	calc8042: LREAL :=  10;
	calc8043: LREAL :=  10;
	calc8044: LREAL :=  10;
	calc8045: LREAL :=  10;
	calc8046: LREAL :=  10;
	calc8047: LREAL :=  10;
	calc8048: LREAL :=  10;
	calc8049: LREAL :=  10;
	calc8050: LREAL :=  10;
	calc8051: LREAL :=  10;
	calc8052: LREAL :=  10;
	calc8053: LREAL :=  10;
	calc8054: LREAL :=  10;
	calc8055: LREAL :=  10;
	calc8056: LREAL :=  10;
	calc8057: LREAL :=  10;
	calc8058: LREAL :=  10;
	calc8059: LREAL :=  10;
	calc8060: LREAL :=  10;
	calc8061: LREAL :=  10;
	calc8062: LREAL :=  10;
	calc8063: LREAL :=  10;
	calc8064: LREAL :=  10;
	calc8065: LREAL :=  10;
	calc8066: LREAL :=  10;
	calc8067: LREAL :=  10;
	calc8068: LREAL :=  10;
	calc8069: LREAL :=  10;
	calc8070: LREAL :=  10;
	calc8071: LREAL :=  10;
	calc8072: LREAL :=  10;
	calc8073: LREAL :=  10;
	calc8074: LREAL :=  10;
	calc8075: LREAL :=  10;
	calc8076: LREAL :=  10;
	calc8077: LREAL :=  10;
	calc8078: LREAL :=  10;
	calc8079: LREAL :=  10;
	calc8080: LREAL :=  10;
	calc8081: LREAL :=  10;
	calc8082: LREAL :=  10;
	calc8083: LREAL :=  10;
	calc8084: LREAL :=  10;
	calc8085: LREAL :=  10;
	calc8086: LREAL :=  10;
	calc8087: LREAL :=  10;
	calc8088: LREAL :=  10;
	calc8089: LREAL :=  10;
	calc8090: LREAL :=  10;
	calc8091: LREAL :=  10;
	calc8092: LREAL :=  10;
	calc8093: LREAL :=  10;
	calc8094: LREAL :=  10;
	calc8095: LREAL :=  10;
	calc8096: LREAL :=  10;
	calc8097: LREAL :=  10;
	calc8098: LREAL :=  10;
	calc8099: LREAL :=  10;
	calc8100: LREAL :=  10;
	calc8101: LREAL :=  10;
	calc8102: LREAL :=  10;
	calc8103: LREAL :=  10;
	calc8104: LREAL :=  10;
	calc8105: LREAL :=  10;
	calc8106: LREAL :=  10;
	calc8107: LREAL :=  10;
	calc8108: LREAL :=  10;
	calc8109: LREAL :=  10;
	calc8110: LREAL :=  10;
	calc8111: LREAL :=  10;
	calc8112: LREAL :=  10;
	calc8113: LREAL :=  10;
	calc8114: LREAL :=  10;
	calc8115: LREAL :=  10;
	calc8116: LREAL :=  10;
	calc8117: LREAL :=  10;
	calc8118: LREAL :=  10;
	calc8119: LREAL :=  10;
	calc8120: LREAL :=  10;
	calc8121: LREAL :=  10;
	calc8122: LREAL :=  10;
	calc8123: LREAL :=  10;
	calc8124: LREAL :=  10;
	calc8125: LREAL :=  10;
	calc8126: LREAL :=  10;
	calc8127: LREAL :=  10;
	calc8128: LREAL :=  10;
	calc8129: LREAL :=  10;
	calc8130: LREAL :=  10;
	calc8131: LREAL :=  10;
	calc8132: LREAL :=  10;
	calc8133: LREAL :=  10;
	calc8134: LREAL :=  10;
	calc8135: LREAL :=  10;
	calc8136: LREAL :=  10;
	calc8137: LREAL :=  10;
	calc8138: LREAL :=  10;
	calc8139: LREAL :=  10;
	calc8140: LREAL :=  10;
	calc8141: LREAL :=  10;
	calc8142: LREAL :=  10;
	calc8143: LREAL :=  10;
	calc8144: LREAL :=  10;
	calc8145: LREAL :=  10;
	calc8146: LREAL :=  10;
	calc8147: LREAL :=  10;
	calc8148: LREAL :=  10;
	calc8149: LREAL :=  10;
	calc8150: LREAL :=  10;
	calc8151: LREAL :=  10;
	calc8152: LREAL :=  10;
	calc8153: LREAL :=  10;
	calc8154: LREAL :=  10;
	calc8155: LREAL :=  10;
	calc8156: LREAL :=  10;
	calc8157: LREAL :=  10;
	calc8158: LREAL :=  10;
	calc8159: LREAL :=  10;
	calc8160: LREAL :=  10;
	calc8161: LREAL :=  10;
	calc8162: LREAL :=  10;
	calc8163: LREAL :=  10;
	calc8164: LREAL :=  10;
	calc8165: LREAL :=  10;
	calc8166: LREAL :=  10;
	calc8167: LREAL :=  10;
	calc8168: LREAL :=  10;
	calc8169: LREAL :=  10;
	calc8170: LREAL :=  10;
	calc8171: LREAL :=  10;
	calc8172: LREAL :=  10;
	calc8173: LREAL :=  10;
	calc8174: LREAL :=  10;
	calc8175: LREAL :=  10;
	calc8176: LREAL :=  10;
	calc8177: LREAL :=  10;
	calc8178: LREAL :=  10;
	calc8179: LREAL :=  10;
	calc8180: LREAL :=  10;
	calc8181: LREAL :=  10;
	calc8182: LREAL :=  10;
	calc8183: LREAL :=  10;
	calc8184: LREAL :=  10;
	calc8185: LREAL :=  10;
	calc8186: LREAL :=  10;
	calc8187: LREAL :=  10;
	calc8188: LREAL :=  10;
	calc8189: LREAL :=  10;
	calc8190: LREAL :=  10;
	calc8191: LREAL :=  10;
	calc8192: LREAL :=  10;
	calc8193: LREAL :=  10;
	calc8194: LREAL :=  10;
	calc8195: LREAL :=  10;
	calc8196: LREAL :=  10;
	calc8197: LREAL :=  10;
	calc8198: LREAL :=  10;
	calc8199: LREAL :=  10;
	calc8200: LREAL :=  10;
	calc8201: LREAL :=  10;
	calc8202: LREAL :=  10;
	calc8203: LREAL :=  10;
	calc8204: LREAL :=  10;
	calc8205: LREAL :=  10;
	calc8206: LREAL :=  10;
	calc8207: LREAL :=  10;
	calc8208: LREAL :=  10;
	calc8209: LREAL :=  10;
	calc8210: LREAL :=  10;
	calc8211: LREAL :=  10;
	calc8212: LREAL :=  10;
	calc8213: LREAL :=  10;
	calc8214: LREAL :=  10;
	calc8215: LREAL :=  10;
	calc8216: LREAL :=  10;
	calc8217: LREAL :=  10;
	calc8218: LREAL :=  10;
	calc8219: LREAL :=  10;
	calc8220: LREAL :=  10;
	calc8221: LREAL :=  10;
	calc8222: LREAL :=  10;
	calc8223: LREAL :=  10;
	calc8224: LREAL :=  10;
	calc8225: LREAL :=  10;
	calc8226: LREAL :=  10;
	calc8227: LREAL :=  10;
	calc8228: LREAL :=  10;
	calc8229: LREAL :=  10;
	calc8230: LREAL :=  10;
	calc8231: LREAL :=  10;
	calc8232: LREAL :=  10;
	calc8233: LREAL :=  10;
	calc8234: LREAL :=  10;
	calc8235: LREAL :=  10;
	calc8236: LREAL :=  10;
	calc8237: LREAL :=  10;
	calc8238: LREAL :=  10;
	calc8239: LREAL :=  10;
	calc8240: LREAL :=  10;
	calc8241: LREAL :=  10;
	calc8242: LREAL :=  10;
	calc8243: LREAL :=  10;
	calc8244: LREAL :=  10;
	calc8245: LREAL :=  10;
	calc8246: LREAL :=  10;
	calc8247: LREAL :=  10;
	calc8248: LREAL :=  10;
	calc8249: LREAL :=  10;
	calc8250: LREAL :=  10;
	calc8251: LREAL :=  10;
	calc8252: LREAL :=  10;
	calc8253: LREAL :=  10;
	calc8254: LREAL :=  10;
	calc8255: LREAL :=  10;
	calc8256: LREAL :=  10;
	calc8257: LREAL :=  10;
	calc8258: LREAL :=  10;
	calc8259: LREAL :=  10;
	calc8260: LREAL :=  10;
	calc8261: LREAL :=  10;
	calc8262: LREAL :=  10;
	calc8263: LREAL :=  10;
	calc8264: LREAL :=  10;
	calc8265: LREAL :=  10;
	calc8266: LREAL :=  10;
	calc8267: LREAL :=  10;
	calc8268: LREAL :=  10;
	calc8269: LREAL :=  10;
	calc8270: LREAL :=  10;
	calc8271: LREAL :=  10;
	calc8272: LREAL :=  10;
	calc8273: LREAL :=  10;
	calc8274: LREAL :=  10;
	calc8275: LREAL :=  10;
	calc8276: LREAL :=  10;
	calc8277: LREAL :=  10;
	calc8278: LREAL :=  10;
	calc8279: LREAL :=  10;
	calc8280: LREAL :=  10;
	calc8281: LREAL :=  10;
	calc8282: LREAL :=  10;
	calc8283: LREAL :=  10;
	calc8284: LREAL :=  10;
	calc8285: LREAL :=  10;
	calc8286: LREAL :=  10;
	calc8287: LREAL :=  10;
	calc8288: LREAL :=  10;
	calc8289: LREAL :=  10;
	calc8290: LREAL :=  10;
	calc8291: LREAL :=  10;
	calc8292: LREAL :=  10;
	calc8293: LREAL :=  10;
	calc8294: LREAL :=  10;
	calc8295: LREAL :=  10;
	calc8296: LREAL :=  10;
	calc8297: LREAL :=  10;
	calc8298: LREAL :=  10;
	calc8299: LREAL :=  10;
	calc8300: LREAL :=  10;
	calc8301: LREAL :=  10;
	calc8302: LREAL :=  10;
	calc8303: LREAL :=  10;
	calc8304: LREAL :=  10;
	calc8305: LREAL :=  10;
	calc8306: LREAL :=  10;
	calc8307: LREAL :=  10;
	calc8308: LREAL :=  10;
	calc8309: LREAL :=  10;
	calc8310: LREAL :=  10;
	calc8311: LREAL :=  10;
	calc8312: LREAL :=  10;
	calc8313: LREAL :=  10;
	calc8314: LREAL :=  10;
	calc8315: LREAL :=  10;
	calc8316: LREAL :=  10;
	calc8317: LREAL :=  10;
	calc8318: LREAL :=  10;
	calc8319: LREAL :=  10;
	calc8320: LREAL :=  10;
	calc8321: LREAL :=  10;
	calc8322: LREAL :=  10;
	calc8323: LREAL :=  10;
	calc8324: LREAL :=  10;
	calc8325: LREAL :=  10;
	calc8326: LREAL :=  10;
	calc8327: LREAL :=  10;
	calc8328: LREAL :=  10;
	calc8329: LREAL :=  10;
	calc8330: LREAL :=  10;
	calc8331: LREAL :=  10;
	calc8332: LREAL :=  10;
	calc8333: LREAL :=  10;
	calc8334: LREAL :=  10;
	calc8335: LREAL :=  10;
	calc8336: LREAL :=  10;
	calc8337: LREAL :=  10;
	calc8338: LREAL :=  10;
	calc8339: LREAL :=  10;
	calc8340: LREAL :=  10;
	calc8341: LREAL :=  10;
	calc8342: LREAL :=  10;
	calc8343: LREAL :=  10;
	calc8344: LREAL :=  10;
	calc8345: LREAL :=  10;
	calc8346: LREAL :=  10;
	calc8347: LREAL :=  10;
	calc8348: LREAL :=  10;
	calc8349: LREAL :=  10;
	calc8350: LREAL :=  10;
	calc8351: LREAL :=  10;
	calc8352: LREAL :=  10;
	calc8353: LREAL :=  10;
	calc8354: LREAL :=  10;
	calc8355: LREAL :=  10;
	calc8356: LREAL :=  10;
	calc8357: LREAL :=  10;
	calc8358: LREAL :=  10;
	calc8359: LREAL :=  10;
	calc8360: LREAL :=  10;
	calc8361: LREAL :=  10;
	calc8362: LREAL :=  10;
	calc8363: LREAL :=  10;
	calc8364: LREAL :=  10;
	calc8365: LREAL :=  10;
	calc8366: LREAL :=  10;
	calc8367: LREAL :=  10;
	calc8368: LREAL :=  10;
	calc8369: LREAL :=  10;
	calc8370: LREAL :=  10;
	calc8371: LREAL :=  10;
	calc8372: LREAL :=  10;
	calc8373: LREAL :=  10;
	calc8374: LREAL :=  10;
	calc8375: LREAL :=  10;
	calc8376: LREAL :=  10;
	calc8377: LREAL :=  10;
	calc8378: LREAL :=  10;
	calc8379: LREAL :=  10;
	calc8380: LREAL :=  10;
	calc8381: LREAL :=  10;
	calc8382: LREAL :=  10;
	calc8383: LREAL :=  10;
	calc8384: LREAL :=  10;
	calc8385: LREAL :=  10;
	calc8386: LREAL :=  10;
	calc8387: LREAL :=  10;
	calc8388: LREAL :=  10;
	calc8389: LREAL :=  10;
	calc8390: LREAL :=  10;
	calc8391: LREAL :=  10;
	calc8392: LREAL :=  10;
	calc8393: LREAL :=  10;
	calc8394: LREAL :=  10;
	calc8395: LREAL :=  10;
	calc8396: LREAL :=  10;
	calc8397: LREAL :=  10;
	calc8398: LREAL :=  10;
	calc8399: LREAL :=  10;
	calc8400: LREAL :=  10;
	calc8401: LREAL :=  10;
	calc8402: LREAL :=  10;
	calc8403: LREAL :=  10;
	calc8404: LREAL :=  10;
	calc8405: LREAL :=  10;
	calc8406: LREAL :=  10;
	calc8407: LREAL :=  10;
	calc8408: LREAL :=  10;
	calc8409: LREAL :=  10;
	calc8410: LREAL :=  10;
	calc8411: LREAL :=  10;
	calc8412: LREAL :=  10;
	calc8413: LREAL :=  10;
	calc8414: LREAL :=  10;
	calc8415: LREAL :=  10;
	calc8416: LREAL :=  10;
	calc8417: LREAL :=  10;
	calc8418: LREAL :=  10;
	calc8419: LREAL :=  10;
	calc8420: LREAL :=  10;
	calc8421: LREAL :=  10;
	calc8422: LREAL :=  10;
	calc8423: LREAL :=  10;
	calc8424: LREAL :=  10;
	calc8425: LREAL :=  10;
	calc8426: LREAL :=  10;
	calc8427: LREAL :=  10;
	calc8428: LREAL :=  10;
	calc8429: LREAL :=  10;
	calc8430: LREAL :=  10;
	calc8431: LREAL :=  10;
	calc8432: LREAL :=  10;
	calc8433: LREAL :=  10;
	calc8434: LREAL :=  10;
	calc8435: LREAL :=  10;
	calc8436: LREAL :=  10;
	calc8437: LREAL :=  10;
	calc8438: LREAL :=  10;
	calc8439: LREAL :=  10;
	calc8440: LREAL :=  10;
	calc8441: LREAL :=  10;
	calc8442: LREAL :=  10;
	calc8443: LREAL :=  10;
	calc8444: LREAL :=  10;
	calc8445: LREAL :=  10;
	calc8446: LREAL :=  10;
	calc8447: LREAL :=  10;
	calc8448: LREAL :=  10;
	calc8449: LREAL :=  10;
	calc8450: LREAL :=  10;
	calc8451: LREAL :=  10;
	calc8452: LREAL :=  10;
	calc8453: LREAL :=  10;
	calc8454: LREAL :=  10;
	calc8455: LREAL :=  10;
	calc8456: LREAL :=  10;
	calc8457: LREAL :=  10;
	calc8458: LREAL :=  10;
	calc8459: LREAL :=  10;
	calc8460: LREAL :=  10;
	calc8461: LREAL :=  10;
	calc8462: LREAL :=  10;
	calc8463: LREAL :=  10;
	calc8464: LREAL :=  10;
	calc8465: LREAL :=  10;
	calc8466: LREAL :=  10;
	calc8467: LREAL :=  10;
	calc8468: LREAL :=  10;
	calc8469: LREAL :=  10;
	calc8470: LREAL :=  10;
	calc8471: LREAL :=  10;
	calc8472: LREAL :=  10;
	calc8473: LREAL :=  10;
	calc8474: LREAL :=  10;
	calc8475: LREAL :=  10;
	calc8476: LREAL :=  10;
	calc8477: LREAL :=  10;
	calc8478: LREAL :=  10;
	calc8479: LREAL :=  10;
	calc8480: LREAL :=  10;
	calc8481: LREAL :=  10;
	calc8482: LREAL :=  10;
	calc8483: LREAL :=  10;
	calc8484: LREAL :=  10;
	calc8485: LREAL :=  10;
	calc8486: LREAL :=  10;
	calc8487: LREAL :=  10;
	calc8488: LREAL :=  10;
	calc8489: LREAL :=  10;
	calc8490: LREAL :=  10;
	calc8491: LREAL :=  10;
	calc8492: LREAL :=  10;
	calc8493: LREAL :=  10;
	calc8494: LREAL :=  10;
	calc8495: LREAL :=  10;
	calc8496: LREAL :=  10;
	calc8497: LREAL :=  10;
	calc8498: LREAL :=  10;
	calc8499: LREAL :=  10;
	calc8500: LREAL :=  10;
	calc8501: LREAL :=  10;
	calc8502: LREAL :=  10;
	calc8503: LREAL :=  10;
	calc8504: LREAL :=  10;
	calc8505: LREAL :=  10;
	calc8506: LREAL :=  10;
	calc8507: LREAL :=  10;
	calc8508: LREAL :=  10;
	calc8509: LREAL :=  10;
	calc8510: LREAL :=  10;
	calc8511: LREAL :=  10;
	calc8512: LREAL :=  10;
	calc8513: LREAL :=  10;
	calc8514: LREAL :=  10;
	calc8515: LREAL :=  10;
	calc8516: LREAL :=  10;
	calc8517: LREAL :=  10;
	calc8518: LREAL :=  10;
	calc8519: LREAL :=  10;
	calc8520: LREAL :=  10;
	calc8521: LREAL :=  10;
	calc8522: LREAL :=  10;
	calc8523: LREAL :=  10;
	calc8524: LREAL :=  10;
	calc8525: LREAL :=  10;
	calc8526: LREAL :=  10;
	calc8527: LREAL :=  10;
	calc8528: LREAL :=  10;
	calc8529: LREAL :=  10;
	calc8530: LREAL :=  10;
	calc8531: LREAL :=  10;
	calc8532: LREAL :=  10;
	calc8533: LREAL :=  10;
	calc8534: LREAL :=  10;
	calc8535: LREAL :=  10;
	calc8536: LREAL :=  10;
	calc8537: LREAL :=  10;
	calc8538: LREAL :=  10;
	calc8539: LREAL :=  10;
	calc8540: LREAL :=  10;
	calc8541: LREAL :=  10;
	calc8542: LREAL :=  10;
	calc8543: LREAL :=  10;
	calc8544: LREAL :=  10;
	calc8545: LREAL :=  10;
	calc8546: LREAL :=  10;
	calc8547: LREAL :=  10;
	calc8548: LREAL :=  10;
	calc8549: LREAL :=  10;
	calc8550: LREAL :=  10;
	calc8551: LREAL :=  10;
	calc8552: LREAL :=  10;
	calc8553: LREAL :=  10;
	calc8554: LREAL :=  10;
	calc8555: LREAL :=  10;
	calc8556: LREAL :=  10;
	calc8557: LREAL :=  10;
	calc8558: LREAL :=  10;
	calc8559: LREAL :=  10;
	calc8560: LREAL :=  10;
	calc8561: LREAL :=  10;
	calc8562: LREAL :=  10;
	calc8563: LREAL :=  10;
	calc8564: LREAL :=  10;
	calc8565: LREAL :=  10;
	calc8566: LREAL :=  10;
	calc8567: LREAL :=  10;
	calc8568: LREAL :=  10;
	calc8569: LREAL :=  10;
	calc8570: LREAL :=  10;
	calc8571: LREAL :=  10;
	calc8572: LREAL :=  10;
	calc8573: LREAL :=  10;
	calc8574: LREAL :=  10;
	calc8575: LREAL :=  10;
	calc8576: LREAL :=  10;
	calc8577: LREAL :=  10;
	calc8578: LREAL :=  10;
	calc8579: LREAL :=  10;
	calc8580: LREAL :=  10;
	calc8581: LREAL :=  10;
	calc8582: LREAL :=  10;
	calc8583: LREAL :=  10;
	calc8584: LREAL :=  10;
	calc8585: LREAL :=  10;
	calc8586: LREAL :=  10;
	calc8587: LREAL :=  10;
	calc8588: LREAL :=  10;
	calc8589: LREAL :=  10;
	calc8590: LREAL :=  10;
	calc8591: LREAL :=  10;
	calc8592: LREAL :=  10;
	calc8593: LREAL :=  10;
	calc8594: LREAL :=  10;
	calc8595: LREAL :=  10;
	calc8596: LREAL :=  10;
	calc8597: LREAL :=  10;
	calc8598: LREAL :=  10;
	calc8599: LREAL :=  10;
	calc8600: LREAL :=  10;
	calc8601: LREAL :=  10;
	calc8602: LREAL :=  10;
	calc8603: LREAL :=  10;
	calc8604: LREAL :=  10;
	calc8605: LREAL :=  10;
	calc8606: LREAL :=  10;
	calc8607: LREAL :=  10;
	calc8608: LREAL :=  10;
	calc8609: LREAL :=  10;
	calc8610: LREAL :=  10;
	calc8611: LREAL :=  10;
	calc8612: LREAL :=  10;
	calc8613: LREAL :=  10;
	calc8614: LREAL :=  10;
	calc8615: LREAL :=  10;
	calc8616: LREAL :=  10;
	calc8617: LREAL :=  10;
	calc8618: LREAL :=  10;
	calc8619: LREAL :=  10;
	calc8620: LREAL :=  10;
	calc8621: LREAL :=  10;
	calc8622: LREAL :=  10;
	calc8623: LREAL :=  10;
	calc8624: LREAL :=  10;
	calc8625: LREAL :=  10;
	calc8626: LREAL :=  10;
	calc8627: LREAL :=  10;
	calc8628: LREAL :=  10;
	calc8629: LREAL :=  10;
	calc8630: LREAL :=  10;
	calc8631: LREAL :=  10;
	calc8632: LREAL :=  10;
	calc8633: LREAL :=  10;
	calc8634: LREAL :=  10;
	calc8635: LREAL :=  10;
	calc8636: LREAL :=  10;
	calc8637: LREAL :=  10;
	calc8638: LREAL :=  10;
	calc8639: LREAL :=  10;
	calc8640: LREAL :=  10;
	calc8641: LREAL :=  10;
	calc8642: LREAL :=  10;
	calc8643: LREAL :=  10;
	calc8644: LREAL :=  10;
	calc8645: LREAL :=  10;
	calc8646: LREAL :=  10;
	calc8647: LREAL :=  10;
	calc8648: LREAL :=  10;
	calc8649: LREAL :=  10;
	calc8650: LREAL :=  10;
	calc8651: LREAL :=  10;
	calc8652: LREAL :=  10;
	calc8653: LREAL :=  10;
	calc8654: LREAL :=  10;
	calc8655: LREAL :=  10;
	calc8656: LREAL :=  10;
	calc8657: LREAL :=  10;
	calc8658: LREAL :=  10;
	calc8659: LREAL :=  10;
	calc8660: LREAL :=  10;
	calc8661: LREAL :=  10;
	calc8662: LREAL :=  10;
	calc8663: LREAL :=  10;
	calc8664: LREAL :=  10;
	calc8665: LREAL :=  10;
	calc8666: LREAL :=  10;
	calc8667: LREAL :=  10;
	calc8668: LREAL :=  10;
	calc8669: LREAL :=  10;
	calc8670: LREAL :=  10;
	calc8671: LREAL :=  10;
	calc8672: LREAL :=  10;
	calc8673: LREAL :=  10;
	calc8674: LREAL :=  10;
	calc8675: LREAL :=  10;
	calc8676: LREAL :=  10;
	calc8677: LREAL :=  10;
	calc8678: LREAL :=  10;
	calc8679: LREAL :=  10;
	calc8680: LREAL :=  10;
	calc8681: LREAL :=  10;
	calc8682: LREAL :=  10;
	calc8683: LREAL :=  10;
	calc8684: LREAL :=  10;
	calc8685: LREAL :=  10;
	calc8686: LREAL :=  10;
	calc8687: LREAL :=  10;
	calc8688: LREAL :=  10;
	calc8689: LREAL :=  10;
	calc8690: LREAL :=  10;
	calc8691: LREAL :=  10;
	calc8692: LREAL :=  10;
	calc8693: LREAL :=  10;
	calc8694: LREAL :=  10;
	calc8695: LREAL :=  10;
	calc8696: LREAL :=  10;
	calc8697: LREAL :=  10;
	calc8698: LREAL :=  10;
	calc8699: LREAL :=  10;
	calc8700: LREAL :=  10;
	calc8701: LREAL :=  10;
	calc8702: LREAL :=  10;
	calc8703: LREAL :=  10;
	calc8704: LREAL :=  10;
	calc8705: LREAL :=  10;
	calc8706: LREAL :=  10;
	calc8707: LREAL :=  10;
	calc8708: LREAL :=  10;
	calc8709: LREAL :=  10;
	calc8710: LREAL :=  10;
	calc8711: LREAL :=  10;
	calc8712: LREAL :=  10;
	calc8713: LREAL :=  10;
	calc8714: LREAL :=  10;
	calc8715: LREAL :=  10;
	calc8716: LREAL :=  10;
	calc8717: LREAL :=  10;
	calc8718: LREAL :=  10;
	calc8719: LREAL :=  10;
	calc8720: LREAL :=  10;
	calc8721: LREAL :=  10;
	calc8722: LREAL :=  10;
	calc8723: LREAL :=  10;
	calc8724: LREAL :=  10;
	calc8725: LREAL :=  10;
	calc8726: LREAL :=  10;
	calc8727: LREAL :=  10;
	calc8728: LREAL :=  10;
	calc8729: LREAL :=  10;
	calc8730: LREAL :=  10;
	calc8731: LREAL :=  10;
	calc8732: LREAL :=  10;
	calc8733: LREAL :=  10;
	calc8734: LREAL :=  10;
	calc8735: LREAL :=  10;
	calc8736: LREAL :=  10;
	calc8737: LREAL :=  10;
	calc8738: LREAL :=  10;
	calc8739: LREAL :=  10;
	calc8740: LREAL :=  10;
	calc8741: LREAL :=  10;
	calc8742: LREAL :=  10;
	calc8743: LREAL :=  10;
	calc8744: LREAL :=  10;
	calc8745: LREAL :=  10;
	calc8746: LREAL :=  10;
	calc8747: LREAL :=  10;
	calc8748: LREAL :=  10;
	calc8749: LREAL :=  10;
	calc8750: LREAL :=  10;
	calc8751: LREAL :=  10;
	calc8752: LREAL :=  10;
	calc8753: LREAL :=  10;
	calc8754: LREAL :=  10;
	calc8755: LREAL :=  10;
	calc8756: LREAL :=  10;
	calc8757: LREAL :=  10;
	calc8758: LREAL :=  10;
	calc8759: LREAL :=  10;
	calc8760: LREAL :=  10;
	calc8761: LREAL :=  10;
	calc8762: LREAL :=  10;
	calc8763: LREAL :=  10;
	calc8764: LREAL :=  10;
	calc8765: LREAL :=  10;
	calc8766: LREAL :=  10;
	calc8767: LREAL :=  10;
	calc8768: LREAL :=  10;
	calc8769: LREAL :=  10;
	calc8770: LREAL :=  10;
	calc8771: LREAL :=  10;
	calc8772: LREAL :=  10;
	calc8773: LREAL :=  10;
	calc8774: LREAL :=  10;
	calc8775: LREAL :=  10;
	calc8776: LREAL :=  10;
	calc8777: LREAL :=  10;
	calc8778: LREAL :=  10;
	calc8779: LREAL :=  10;
	calc8780: LREAL :=  10;
	calc8781: LREAL :=  10;
	calc8782: LREAL :=  10;
	calc8783: LREAL :=  10;
	calc8784: LREAL :=  10;
	calc8785: LREAL :=  10;
	calc8786: LREAL :=  10;
	calc8787: LREAL :=  10;
	calc8788: LREAL :=  10;
	calc8789: LREAL :=  10;
	calc8790: LREAL :=  10;
	calc8791: LREAL :=  10;
	calc8792: LREAL :=  10;
	calc8793: LREAL :=  10;
	calc8794: LREAL :=  10;
	calc8795: LREAL :=  10;
	calc8796: LREAL :=  10;
	calc8797: LREAL :=  10;
	calc8798: LREAL :=  10;
	calc8799: LREAL :=  10;
	calc8800: LREAL :=  10;
	calc8801: LREAL :=  10;
	calc8802: LREAL :=  10;
	calc8803: LREAL :=  10;
	calc8804: LREAL :=  10;
	calc8805: LREAL :=  10;
	calc8806: LREAL :=  10;
	calc8807: LREAL :=  10;
	calc8808: LREAL :=  10;
	calc8809: LREAL :=  10;
	calc8810: LREAL :=  10;
	calc8811: LREAL :=  10;
	calc8812: LREAL :=  10;
	calc8813: LREAL :=  10;
	calc8814: LREAL :=  10;
	calc8815: LREAL :=  10;
	calc8816: LREAL :=  10;
	calc8817: LREAL :=  10;
	calc8818: LREAL :=  10;
	calc8819: LREAL :=  10;
	calc8820: LREAL :=  10;
	calc8821: LREAL :=  10;
	calc8822: LREAL :=  10;
	calc8823: LREAL :=  10;
	calc8824: LREAL :=  10;
	calc8825: LREAL :=  10;
	calc8826: LREAL :=  10;
	calc8827: LREAL :=  10;
	calc8828: LREAL :=  10;
	calc8829: LREAL :=  10;
	calc8830: LREAL :=  10;
	calc8831: LREAL :=  10;
	calc8832: LREAL :=  10;
	calc8833: LREAL :=  10;
	calc8834: LREAL :=  10;
	calc8835: LREAL :=  10;
	calc8836: LREAL :=  10;
	calc8837: LREAL :=  10;
	calc8838: LREAL :=  10;
	calc8839: LREAL :=  10;
	calc8840: LREAL :=  10;
	calc8841: LREAL :=  10;
	calc8842: LREAL :=  10;
	calc8843: LREAL :=  10;
	calc8844: LREAL :=  10;
	calc8845: LREAL :=  10;
	calc8846: LREAL :=  10;
	calc8847: LREAL :=  10;
	calc8848: LREAL :=  10;
	calc8849: LREAL :=  10;
	calc8850: LREAL :=  10;
	calc8851: LREAL :=  10;
	calc8852: LREAL :=  10;
	calc8853: LREAL :=  10;
	calc8854: LREAL :=  10;
	calc8855: LREAL :=  10;
	calc8856: LREAL :=  10;
	calc8857: LREAL :=  10;
	calc8858: LREAL :=  10;
	calc8859: LREAL :=  10;
	calc8860: LREAL :=  10;
	calc8861: LREAL :=  10;
	calc8862: LREAL :=  10;
	calc8863: LREAL :=  10;
	calc8864: LREAL :=  10;
	calc8865: LREAL :=  10;
	calc8866: LREAL :=  10;
	calc8867: LREAL :=  10;
	calc8868: LREAL :=  10;
	calc8869: LREAL :=  10;
	calc8870: LREAL :=  10;
	calc8871: LREAL :=  10;
	calc8872: LREAL :=  10;
	calc8873: LREAL :=  10;
	calc8874: LREAL :=  10;
	calc8875: LREAL :=  10;
	calc8876: LREAL :=  10;
	calc8877: LREAL :=  10;
	calc8878: LREAL :=  10;
	calc8879: LREAL :=  10;
	calc8880: LREAL :=  10;
	calc8881: LREAL :=  10;
	calc8882: LREAL :=  10;
	calc8883: LREAL :=  10;
	calc8884: LREAL :=  10;
	calc8885: LREAL :=  10;
	calc8886: LREAL :=  10;
	calc8887: LREAL :=  10;
	calc8888: LREAL :=  10;
	calc8889: LREAL :=  10;
	calc8890: LREAL :=  10;
	calc8891: LREAL :=  10;
	calc8892: LREAL :=  10;
	calc8893: LREAL :=  10;
	calc8894: LREAL :=  10;
	calc8895: LREAL :=  10;
	calc8896: LREAL :=  10;
	calc8897: LREAL :=  10;
	calc8898: LREAL :=  10;
	calc8899: LREAL :=  10;
	calc8900: LREAL :=  10;
	calc8901: LREAL :=  10;
	calc8902: LREAL :=  10;
	calc8903: LREAL :=  10;
	calc8904: LREAL :=  10;
	calc8905: LREAL :=  10;
	calc8906: LREAL :=  10;
	calc8907: LREAL :=  10;
	calc8908: LREAL :=  10;
	calc8909: LREAL :=  10;
	calc8910: LREAL :=  10;
	calc8911: LREAL :=  10;
	calc8912: LREAL :=  10;
	calc8913: LREAL :=  10;
	calc8914: LREAL :=  10;
	calc8915: LREAL :=  10;
	calc8916: LREAL :=  10;
	calc8917: LREAL :=  10;
	calc8918: LREAL :=  10;
	calc8919: LREAL :=  10;
	calc8920: LREAL :=  10;
	calc8921: LREAL :=  10;
	calc8922: LREAL :=  10;
	calc8923: LREAL :=  10;
	calc8924: LREAL :=  10;
	calc8925: LREAL :=  10;
	calc8926: LREAL :=  10;
	calc8927: LREAL :=  10;
	calc8928: LREAL :=  10;
	calc8929: LREAL :=  10;
	calc8930: LREAL :=  10;
	calc8931: LREAL :=  10;
	calc8932: LREAL :=  10;
	calc8933: LREAL :=  10;
	calc8934: LREAL :=  10;
	calc8935: LREAL :=  10;
	calc8936: LREAL :=  10;
	calc8937: LREAL :=  10;
	calc8938: LREAL :=  10;
	calc8939: LREAL :=  10;
	calc8940: LREAL :=  10;
	calc8941: LREAL :=  10;
	calc8942: LREAL :=  10;
	calc8943: LREAL :=  10;
	calc8944: LREAL :=  10;
	calc8945: LREAL :=  10;
	calc8946: LREAL :=  10;
	calc8947: LREAL :=  10;
	calc8948: LREAL :=  10;
	calc8949: LREAL :=  10;
	calc8950: LREAL :=  10;
	calc8951: LREAL :=  10;
	calc8952: LREAL :=  10;
	calc8953: LREAL :=  10;
	calc8954: LREAL :=  10;
	calc8955: LREAL :=  10;
	calc8956: LREAL :=  10;
	calc8957: LREAL :=  10;
	calc8958: LREAL :=  10;
	calc8959: LREAL :=  10;
	calc8960: LREAL :=  10;
	calc8961: LREAL :=  10;
	calc8962: LREAL :=  10;
	calc8963: LREAL :=  10;
	calc8964: LREAL :=  10;
	calc8965: LREAL :=  10;
	calc8966: LREAL :=  10;
	calc8967: LREAL :=  10;
	calc8968: LREAL :=  10;
	calc8969: LREAL :=  10;
	calc8970: LREAL :=  10;
	calc8971: LREAL :=  10;
	calc8972: LREAL :=  10;
	calc8973: LREAL :=  10;
	calc8974: LREAL :=  10;
	calc8975: LREAL :=  10;
	calc8976: LREAL :=  10;
	calc8977: LREAL :=  10;
	calc8978: LREAL :=  10;
	calc8979: LREAL :=  10;
	calc8980: LREAL :=  10;
	calc8981: LREAL :=  10;
	calc8982: LREAL :=  10;
	calc8983: LREAL :=  10;
	calc8984: LREAL :=  10;
	calc8985: LREAL :=  10;
	calc8986: LREAL :=  10;
	calc8987: LREAL :=  10;
	calc8988: LREAL :=  10;
	calc8989: LREAL :=  10;
	calc8990: LREAL :=  10;
	calc8991: LREAL :=  10;
	calc8992: LREAL :=  10;
	calc8993: LREAL :=  10;
	calc8994: LREAL :=  10;
	calc8995: LREAL :=  10;
	calc8996: LREAL :=  10;
	calc8997: LREAL :=  10;
	calc8998: LREAL :=  10;
	calc8999: LREAL :=  10;
	calc9000: LREAL :=  10;
	calc9001: LREAL :=  10;
	calc9002: LREAL :=  10;
	calc9003: LREAL :=  10;
	calc9004: LREAL :=  10;
	calc9005: LREAL :=  10;
	calc9006: LREAL :=  10;
	calc9007: LREAL :=  10;
	calc9008: LREAL :=  10;
	calc9009: LREAL :=  10;
	calc9010: LREAL :=  10;
	calc9011: LREAL :=  10;
	calc9012: LREAL :=  10;
	calc9013: LREAL :=  10;
	calc9014: LREAL :=  10;
	calc9015: LREAL :=  10;
	calc9016: LREAL :=  10;
	calc9017: LREAL :=  10;
	calc9018: LREAL :=  10;
	calc9019: LREAL :=  10;
	calc9020: LREAL :=  10;
	calc9021: LREAL :=  10;
	calc9022: LREAL :=  10;
	calc9023: LREAL :=  10;
	calc9024: LREAL :=  10;
	calc9025: LREAL :=  10;
	calc9026: LREAL :=  10;
	calc9027: LREAL :=  10;
	calc9028: LREAL :=  10;
	calc9029: LREAL :=  10;
	calc9030: LREAL :=  10;
	calc9031: LREAL :=  10;
	calc9032: LREAL :=  10;
	calc9033: LREAL :=  10;
	calc9034: LREAL :=  10;
	calc9035: LREAL :=  10;
	calc9036: LREAL :=  10;
	calc9037: LREAL :=  10;
	calc9038: LREAL :=  10;
	calc9039: LREAL :=  10;
	calc9040: LREAL :=  10;
	calc9041: LREAL :=  10;
	calc9042: LREAL :=  10;
	calc9043: LREAL :=  10;
	calc9044: LREAL :=  10;
	calc9045: LREAL :=  10;
	calc9046: LREAL :=  10;
	calc9047: LREAL :=  10;
	calc9048: LREAL :=  10;
	calc9049: LREAL :=  10;
	calc9050: LREAL :=  10;
	calc9051: LREAL :=  10;
	calc9052: LREAL :=  10;
	calc9053: LREAL :=  10;
	calc9054: LREAL :=  10;
	calc9055: LREAL :=  10;
	calc9056: LREAL :=  10;
	calc9057: LREAL :=  10;
	calc9058: LREAL :=  10;
	calc9059: LREAL :=  10;
	calc9060: LREAL :=  10;
	calc9061: LREAL :=  10;
	calc9062: LREAL :=  10;
	calc9063: LREAL :=  10;
	calc9064: LREAL :=  10;
	calc9065: LREAL :=  10;
	calc9066: LREAL :=  10;
	calc9067: LREAL :=  10;
	calc9068: LREAL :=  10;
	calc9069: LREAL :=  10;
	calc9070: LREAL :=  10;
	calc9071: LREAL :=  10;
	calc9072: LREAL :=  10;
	calc9073: LREAL :=  10;
	calc9074: LREAL :=  10;
	calc9075: LREAL :=  10;
	calc9076: LREAL :=  10;
	calc9077: LREAL :=  10;
	calc9078: LREAL :=  10;
	calc9079: LREAL :=  10;
	calc9080: LREAL :=  10;
	calc9081: LREAL :=  10;
	calc9082: LREAL :=  10;
	calc9083: LREAL :=  10;
	calc9084: LREAL :=  10;
	calc9085: LREAL :=  10;
	calc9086: LREAL :=  10;
	calc9087: LREAL :=  10;
	calc9088: LREAL :=  10;
	calc9089: LREAL :=  10;
	calc9090: LREAL :=  10;
	calc9091: LREAL :=  10;
	calc9092: LREAL :=  10;
	calc9093: LREAL :=  10;
	calc9094: LREAL :=  10;
	calc9095: LREAL :=  10;
	calc9096: LREAL :=  10;
	calc9097: LREAL :=  10;
	calc9098: LREAL :=  10;
	calc9099: LREAL :=  10;
	calc9100: LREAL :=  10;
	calc9101: LREAL :=  10;
	calc9102: LREAL :=  10;
	calc9103: LREAL :=  10;
	calc9104: LREAL :=  10;
	calc9105: LREAL :=  10;
	calc9106: LREAL :=  10;
	calc9107: LREAL :=  10;
	calc9108: LREAL :=  10;
	calc9109: LREAL :=  10;
	calc9110: LREAL :=  10;
	calc9111: LREAL :=  10;
	calc9112: LREAL :=  10;
	calc9113: LREAL :=  10;
	calc9114: LREAL :=  10;
	calc9115: LREAL :=  10;
	calc9116: LREAL :=  10;
	calc9117: LREAL :=  10;
	calc9118: LREAL :=  10;
	calc9119: LREAL :=  10;
	calc9120: LREAL :=  10;
	calc9121: LREAL :=  10;
	calc9122: LREAL :=  10;
	calc9123: LREAL :=  10;
	calc9124: LREAL :=  10;
	calc9125: LREAL :=  10;
	calc9126: LREAL :=  10;
	calc9127: LREAL :=  10;
	calc9128: LREAL :=  10;
	calc9129: LREAL :=  10;
	calc9130: LREAL :=  10;
	calc9131: LREAL :=  10;
	calc9132: LREAL :=  10;
	calc9133: LREAL :=  10;
	calc9134: LREAL :=  10;
	calc9135: LREAL :=  10;
	calc9136: LREAL :=  10;
	calc9137: LREAL :=  10;
	calc9138: LREAL :=  10;
	calc9139: LREAL :=  10;
	calc9140: LREAL :=  10;
	calc9141: LREAL :=  10;
	calc9142: LREAL :=  10;
	calc9143: LREAL :=  10;
	calc9144: LREAL :=  10;
	calc9145: LREAL :=  10;
	calc9146: LREAL :=  10;
	calc9147: LREAL :=  10;
	calc9148: LREAL :=  10;
	calc9149: LREAL :=  10;
	calc9150: LREAL :=  10;
	calc9151: LREAL :=  10;
	calc9152: LREAL :=  10;
	calc9153: LREAL :=  10;
	calc9154: LREAL :=  10;
	calc9155: LREAL :=  10;
	calc9156: LREAL :=  10;
	calc9157: LREAL :=  10;
	calc9158: LREAL :=  10;
	calc9159: LREAL :=  10;
	calc9160: LREAL :=  10;
	calc9161: LREAL :=  10;
	calc9162: LREAL :=  10;
	calc9163: LREAL :=  10;
	calc9164: LREAL :=  10;
	calc9165: LREAL :=  10;
	calc9166: LREAL :=  10;
	calc9167: LREAL :=  10;
	calc9168: LREAL :=  10;
	calc9169: LREAL :=  10;
	calc9170: LREAL :=  10;
	calc9171: LREAL :=  10;
	calc9172: LREAL :=  10;
	calc9173: LREAL :=  10;
	calc9174: LREAL :=  10;
	calc9175: LREAL :=  10;
	calc9176: LREAL :=  10;
	calc9177: LREAL :=  10;
	calc9178: LREAL :=  10;
	calc9179: LREAL :=  10;
	calc9180: LREAL :=  10;
	calc9181: LREAL :=  10;
	calc9182: LREAL :=  10;
	calc9183: LREAL :=  10;
	calc9184: LREAL :=  10;
	calc9185: LREAL :=  10;
	calc9186: LREAL :=  10;
	calc9187: LREAL :=  10;
	calc9188: LREAL :=  10;
	calc9189: LREAL :=  10;
	calc9190: LREAL :=  10;
	calc9191: LREAL :=  10;
	calc9192: LREAL :=  10;
	calc9193: LREAL :=  10;
	calc9194: LREAL :=  10;
	calc9195: LREAL :=  10;
	calc9196: LREAL :=  10;
	calc9197: LREAL :=  10;
	calc9198: LREAL :=  10;
	calc9199: LREAL :=  10;
	calc9200: LREAL :=  10;
	calc9201: LREAL :=  10;
	calc9202: LREAL :=  10;
	calc9203: LREAL :=  10;
	calc9204: LREAL :=  10;
	calc9205: LREAL :=  10;
	calc9206: LREAL :=  10;
	calc9207: LREAL :=  10;
	calc9208: LREAL :=  10;
	calc9209: LREAL :=  10;
	calc9210: LREAL :=  10;
	calc9211: LREAL :=  10;
	calc9212: LREAL :=  10;
	calc9213: LREAL :=  10;
	calc9214: LREAL :=  10;
	calc9215: LREAL :=  10;
	calc9216: LREAL :=  10;
	calc9217: LREAL :=  10;
	calc9218: LREAL :=  10;
	calc9219: LREAL :=  10;
	calc9220: LREAL :=  10;
	calc9221: LREAL :=  10;
	calc9222: LREAL :=  10;
	calc9223: LREAL :=  10;
	calc9224: LREAL :=  10;
	calc9225: LREAL :=  10;
	calc9226: LREAL :=  10;
	calc9227: LREAL :=  10;
	calc9228: LREAL :=  10;
	calc9229: LREAL :=  10;
	calc9230: LREAL :=  10;
	calc9231: LREAL :=  10;
	calc9232: LREAL :=  10;
	calc9233: LREAL :=  10;
	calc9234: LREAL :=  10;
	calc9235: LREAL :=  10;
	calc9236: LREAL :=  10;
	calc9237: LREAL :=  10;
	calc9238: LREAL :=  10;
	calc9239: LREAL :=  10;
	calc9240: LREAL :=  10;
	calc9241: LREAL :=  10;
	calc9242: LREAL :=  10;
	calc9243: LREAL :=  10;
	calc9244: LREAL :=  10;
	calc9245: LREAL :=  10;
	calc9246: LREAL :=  10;
	calc9247: LREAL :=  10;
	calc9248: LREAL :=  10;
	calc9249: LREAL :=  10;
	calc9250: LREAL :=  10;
	calc9251: LREAL :=  10;
	calc9252: LREAL :=  10;
	calc9253: LREAL :=  10;
	calc9254: LREAL :=  10;
	calc9255: LREAL :=  10;
	calc9256: LREAL :=  10;
	calc9257: LREAL :=  10;
	calc9258: LREAL :=  10;
	calc9259: LREAL :=  10;
	calc9260: LREAL :=  10;
	calc9261: LREAL :=  10;
	calc9262: LREAL :=  10;
	calc9263: LREAL :=  10;
	calc9264: LREAL :=  10;
	calc9265: LREAL :=  10;
	calc9266: LREAL :=  10;
	calc9267: LREAL :=  10;
	calc9268: LREAL :=  10;
	calc9269: LREAL :=  10;
	calc9270: LREAL :=  10;
	calc9271: LREAL :=  10;
	calc9272: LREAL :=  10;
	calc9273: LREAL :=  10;
	calc9274: LREAL :=  10;
	calc9275: LREAL :=  10;
	calc9276: LREAL :=  10;
	calc9277: LREAL :=  10;
	calc9278: LREAL :=  10;
	calc9279: LREAL :=  10;
	calc9280: LREAL :=  10;
	calc9281: LREAL :=  10;
	calc9282: LREAL :=  10;
	calc9283: LREAL :=  10;
	calc9284: LREAL :=  10;
	calc9285: LREAL :=  10;
	calc9286: LREAL :=  10;
	calc9287: LREAL :=  10;
	calc9288: LREAL :=  10;
	calc9289: LREAL :=  10;
	calc9290: LREAL :=  10;
	calc9291: LREAL :=  10;
	calc9292: LREAL :=  10;
	calc9293: LREAL :=  10;
	calc9294: LREAL :=  10;
	calc9295: LREAL :=  10;
	calc9296: LREAL :=  10;
	calc9297: LREAL :=  10;
	calc9298: LREAL :=  10;
	calc9299: LREAL :=  10;
	calc9300: LREAL :=  10;
	calc9301: LREAL :=  10;
	calc9302: LREAL :=  10;
	calc9303: LREAL :=  10;
	calc9304: LREAL :=  10;
	calc9305: LREAL :=  10;
	calc9306: LREAL :=  10;
	calc9307: LREAL :=  10;
	calc9308: LREAL :=  10;
	calc9309: LREAL :=  10;
	calc9310: LREAL :=  10;
	calc9311: LREAL :=  10;
	calc9312: LREAL :=  10;
	calc9313: LREAL :=  10;
	calc9314: LREAL :=  10;
	calc9315: LREAL :=  10;
	calc9316: LREAL :=  10;
	calc9317: LREAL :=  10;
	calc9318: LREAL :=  10;
	calc9319: LREAL :=  10;
	calc9320: LREAL :=  10;
	calc9321: LREAL :=  10;
	calc9322: LREAL :=  10;
	calc9323: LREAL :=  10;
	calc9324: LREAL :=  10;
	calc9325: LREAL :=  10;
	calc9326: LREAL :=  10;
	calc9327: LREAL :=  10;
	calc9328: LREAL :=  10;
	calc9329: LREAL :=  10;
	calc9330: LREAL :=  10;
	calc9331: LREAL :=  10;
	calc9332: LREAL :=  10;
	calc9333: LREAL :=  10;
	calc9334: LREAL :=  10;
	calc9335: LREAL :=  10;
	calc9336: LREAL :=  10;
	calc9337: LREAL :=  10;
	calc9338: LREAL :=  10;
	calc9339: LREAL :=  10;
	calc9340: LREAL :=  10;
	calc9341: LREAL :=  10;
	calc9342: LREAL :=  10;
	calc9343: LREAL :=  10;
	calc9344: LREAL :=  10;
	calc9345: LREAL :=  10;
	calc9346: LREAL :=  10;
	calc9347: LREAL :=  10;
	calc9348: LREAL :=  10;
	calc9349: LREAL :=  10;
	calc9350: LREAL :=  10;
	calc9351: LREAL :=  10;
	calc9352: LREAL :=  10;
	calc9353: LREAL :=  10;
	calc9354: LREAL :=  10;
	calc9355: LREAL :=  10;
	calc9356: LREAL :=  10;
	calc9357: LREAL :=  10;
	calc9358: LREAL :=  10;
	calc9359: LREAL :=  10;
	calc9360: LREAL :=  10;
	calc9361: LREAL :=  10;
	calc9362: LREAL :=  10;
	calc9363: LREAL :=  10;
	calc9364: LREAL :=  10;
	calc9365: LREAL :=  10;
	calc9366: LREAL :=  10;
	calc9367: LREAL :=  10;
	calc9368: LREAL :=  10;
	calc9369: LREAL :=  10;
	calc9370: LREAL :=  10;
	calc9371: LREAL :=  10;
	calc9372: LREAL :=  10;
	calc9373: LREAL :=  10;
	calc9374: LREAL :=  10;
	calc9375: LREAL :=  10;
	calc9376: LREAL :=  10;
	calc9377: LREAL :=  10;
	calc9378: LREAL :=  10;
	calc9379: LREAL :=  10;
	calc9380: LREAL :=  10;
	calc9381: LREAL :=  10;
	calc9382: LREAL :=  10;
	calc9383: LREAL :=  10;
	calc9384: LREAL :=  10;
	calc9385: LREAL :=  10;
	calc9386: LREAL :=  10;
	calc9387: LREAL :=  10;
	calc9388: LREAL :=  10;
	calc9389: LREAL :=  10;
	calc9390: LREAL :=  10;
	calc9391: LREAL :=  10;
	calc9392: LREAL :=  10;
	calc9393: LREAL :=  10;
	calc9394: LREAL :=  10;
	calc9395: LREAL :=  10;
	calc9396: LREAL :=  10;
	calc9397: LREAL :=  10;
	calc9398: LREAL :=  10;
	calc9399: LREAL :=  10;
	calc9400: LREAL :=  10;
	calc9401: LREAL :=  10;
	calc9402: LREAL :=  10;
	calc9403: LREAL :=  10;
	calc9404: LREAL :=  10;
	calc9405: LREAL :=  10;
	calc9406: LREAL :=  10;
	calc9407: LREAL :=  10;
	calc9408: LREAL :=  10;
	calc9409: LREAL :=  10;
	calc9410: LREAL :=  10;
	calc9411: LREAL :=  10;
	calc9412: LREAL :=  10;
	calc9413: LREAL :=  10;
	calc9414: LREAL :=  10;
	calc9415: LREAL :=  10;
	calc9416: LREAL :=  10;
	calc9417: LREAL :=  10;
	calc9418: LREAL :=  10;
	calc9419: LREAL :=  10;
	calc9420: LREAL :=  10;
	calc9421: LREAL :=  10;
	calc9422: LREAL :=  10;
	calc9423: LREAL :=  10;
	calc9424: LREAL :=  10;
	calc9425: LREAL :=  10;
	calc9426: LREAL :=  10;
	calc9427: LREAL :=  10;
	calc9428: LREAL :=  10;
	calc9429: LREAL :=  10;
	calc9430: LREAL :=  10;
	calc9431: LREAL :=  10;
	calc9432: LREAL :=  10;
	calc9433: LREAL :=  10;
	calc9434: LREAL :=  10;
	calc9435: LREAL :=  10;
	calc9436: LREAL :=  10;
	calc9437: LREAL :=  10;
	calc9438: LREAL :=  10;
	calc9439: LREAL :=  10;
	calc9440: LREAL :=  10;
	calc9441: LREAL :=  10;
	calc9442: LREAL :=  10;
	calc9443: LREAL :=  10;
	calc9444: LREAL :=  10;
	calc9445: LREAL :=  10;
	calc9446: LREAL :=  10;
	calc9447: LREAL :=  10;
	calc9448: LREAL :=  10;
	calc9449: LREAL :=  10;
	calc9450: LREAL :=  10;
	calc9451: LREAL :=  10;
	calc9452: LREAL :=  10;
	calc9453: LREAL :=  10;
	calc9454: LREAL :=  10;
	calc9455: LREAL :=  10;
	calc9456: LREAL :=  10;
	calc9457: LREAL :=  10;
	calc9458: LREAL :=  10;
	calc9459: LREAL :=  10;
	calc9460: LREAL :=  10;
	calc9461: LREAL :=  10;
	calc9462: LREAL :=  10;
	calc9463: LREAL :=  10;
	calc9464: LREAL :=  10;
	calc9465: LREAL :=  10;
	calc9466: LREAL :=  10;
	calc9467: LREAL :=  10;
	calc9468: LREAL :=  10;
	calc9469: LREAL :=  10;
	calc9470: LREAL :=  10;
	calc9471: LREAL :=  10;
	calc9472: LREAL :=  10;
	calc9473: LREAL :=  10;
	calc9474: LREAL :=  10;
	calc9475: LREAL :=  10;
	calc9476: LREAL :=  10;
	calc9477: LREAL :=  10;
	calc9478: LREAL :=  10;
	calc9479: LREAL :=  10;
	calc9480: LREAL :=  10;
	calc9481: LREAL :=  10;
	calc9482: LREAL :=  10;
	calc9483: LREAL :=  10;
	calc9484: LREAL :=  10;
	calc9485: LREAL :=  10;
	calc9486: LREAL :=  10;
	calc9487: LREAL :=  10;
	calc9488: LREAL :=  10;
	calc9489: LREAL :=  10;
	calc9490: LREAL :=  10;
	calc9491: LREAL :=  10;
	calc9492: LREAL :=  10;
	calc9493: LREAL :=  10;
	calc9494: LREAL :=  10;
	calc9495: LREAL :=  10;
	calc9496: LREAL :=  10;
	calc9497: LREAL :=  10;
	calc9498: LREAL :=  10;
	calc9499: LREAL :=  10;
	calc9500: LREAL :=  10;
	calc9501: LREAL :=  10;
	calc9502: LREAL :=  10;
	calc9503: LREAL :=  10;
	calc9504: LREAL :=  10;
	calc9505: LREAL :=  10;
	calc9506: LREAL :=  10;
	calc9507: LREAL :=  10;
	calc9508: LREAL :=  10;
	calc9509: LREAL :=  10;
	calc9510: LREAL :=  10;
	calc9511: LREAL :=  10;
	calc9512: LREAL :=  10;
	calc9513: LREAL :=  10;
	calc9514: LREAL :=  10;
	calc9515: LREAL :=  10;
	calc9516: LREAL :=  10;
	calc9517: LREAL :=  10;
	calc9518: LREAL :=  10;
	calc9519: LREAL :=  10;
	calc9520: LREAL :=  10;
	calc9521: LREAL :=  10;
	calc9522: LREAL :=  10;
	calc9523: LREAL :=  10;
	calc9524: LREAL :=  10;
	calc9525: LREAL :=  10;
	calc9526: LREAL :=  10;
	calc9527: LREAL :=  10;
	calc9528: LREAL :=  10;
	calc9529: LREAL :=  10;
	calc9530: LREAL :=  10;
	calc9531: LREAL :=  10;
	calc9532: LREAL :=  10;
	calc9533: LREAL :=  10;
	calc9534: LREAL :=  10;
	calc9535: LREAL :=  10;
	calc9536: LREAL :=  10;
	calc9537: LREAL :=  10;
	calc9538: LREAL :=  10;
	calc9539: LREAL :=  10;
	calc9540: LREAL :=  10;
	calc9541: LREAL :=  10;
	calc9542: LREAL :=  10;
	calc9543: LREAL :=  10;
	calc9544: LREAL :=  10;
	calc9545: LREAL :=  10;
	calc9546: LREAL :=  10;
	calc9547: LREAL :=  10;
	calc9548: LREAL :=  10;
	calc9549: LREAL :=  10;
	calc9550: LREAL :=  10;
	calc9551: LREAL :=  10;
	calc9552: LREAL :=  10;
	calc9553: LREAL :=  10;
	calc9554: LREAL :=  10;
	calc9555: LREAL :=  10;
	calc9556: LREAL :=  10;
	calc9557: LREAL :=  10;
	calc9558: LREAL :=  10;
	calc9559: LREAL :=  10;
	calc9560: LREAL :=  10;
	calc9561: LREAL :=  10;
	calc9562: LREAL :=  10;
	calc9563: LREAL :=  10;
	calc9564: LREAL :=  10;
	calc9565: LREAL :=  10;
	calc9566: LREAL :=  10;
	calc9567: LREAL :=  10;
	calc9568: LREAL :=  10;
	calc9569: LREAL :=  10;
	calc9570: LREAL :=  10;
	calc9571: LREAL :=  10;
	calc9572: LREAL :=  10;
	calc9573: LREAL :=  10;
	calc9574: LREAL :=  10;
	calc9575: LREAL :=  10;
	calc9576: LREAL :=  10;
	calc9577: LREAL :=  10;
	calc9578: LREAL :=  10;
	calc9579: LREAL :=  10;
	calc9580: LREAL :=  10;
	calc9581: LREAL :=  10;
	calc9582: LREAL :=  10;
	calc9583: LREAL :=  10;
	calc9584: LREAL :=  10;
	calc9585: LREAL :=  10;
	calc9586: LREAL :=  10;
	calc9587: LREAL :=  10;
	calc9588: LREAL :=  10;
	calc9589: LREAL :=  10;
	calc9590: LREAL :=  10;
	calc9591: LREAL :=  10;
	calc9592: LREAL :=  10;
	calc9593: LREAL :=  10;
	calc9594: LREAL :=  10;
	calc9595: LREAL :=  10;
	calc9596: LREAL :=  10;
	calc9597: LREAL :=  10;
	calc9598: LREAL :=  10;
	calc9599: LREAL :=  10;
	calc9600: LREAL :=  10;
	calc9601: LREAL :=  10;
	calc9602: LREAL :=  10;
	calc9603: LREAL :=  10;
	calc9604: LREAL :=  10;
	calc9605: LREAL :=  10;
	calc9606: LREAL :=  10;
	calc9607: LREAL :=  10;
	calc9608: LREAL :=  10;
	calc9609: LREAL :=  10;
	calc9610: LREAL :=  10;
	calc9611: LREAL :=  10;
	calc9612: LREAL :=  10;
	calc9613: LREAL :=  10;
	calc9614: LREAL :=  10;
	calc9615: LREAL :=  10;
	calc9616: LREAL :=  10;
	calc9617: LREAL :=  10;
	calc9618: LREAL :=  10;
	calc9619: LREAL :=  10;
	calc9620: LREAL :=  10;
	calc9621: LREAL :=  10;
	calc9622: LREAL :=  10;
	calc9623: LREAL :=  10;
	calc9624: LREAL :=  10;
	calc9625: LREAL :=  10;
	calc9626: LREAL :=  10;
	calc9627: LREAL :=  10;
	calc9628: LREAL :=  10;
	calc9629: LREAL :=  10;
	calc9630: LREAL :=  10;
	calc9631: LREAL :=  10;
	calc9632: LREAL :=  10;
	calc9633: LREAL :=  10;
	calc9634: LREAL :=  10;
	calc9635: LREAL :=  10;
	calc9636: LREAL :=  10;
	calc9637: LREAL :=  10;
	calc9638: LREAL :=  10;
	calc9639: LREAL :=  10;
	calc9640: LREAL :=  10;
	calc9641: LREAL :=  10;
	calc9642: LREAL :=  10;
	calc9643: LREAL :=  10;
	calc9644: LREAL :=  10;
	calc9645: LREAL :=  10;
	calc9646: LREAL :=  10;
	calc9647: LREAL :=  10;
	calc9648: LREAL :=  10;
	calc9649: LREAL :=  10;
	calc9650: LREAL :=  10;
	calc9651: LREAL :=  10;
	calc9652: LREAL :=  10;
	calc9653: LREAL :=  10;
	calc9654: LREAL :=  10;
	calc9655: LREAL :=  10;
	calc9656: LREAL :=  10;
	calc9657: LREAL :=  10;
	calc9658: LREAL :=  10;
	calc9659: LREAL :=  10;
	calc9660: LREAL :=  10;
	calc9661: LREAL :=  10;
	calc9662: LREAL :=  10;
	calc9663: LREAL :=  10;
	calc9664: LREAL :=  10;
	calc9665: LREAL :=  10;
	calc9666: LREAL :=  10;
	calc9667: LREAL :=  10;
	calc9668: LREAL :=  10;
	calc9669: LREAL :=  10;
	calc9670: LREAL :=  10;
	calc9671: LREAL :=  10;
	calc9672: LREAL :=  10;
	calc9673: LREAL :=  10;
	calc9674: LREAL :=  10;
	calc9675: LREAL :=  10;
	calc9676: LREAL :=  10;
	calc9677: LREAL :=  10;
	calc9678: LREAL :=  10;
	calc9679: LREAL :=  10;
	calc9680: LREAL :=  10;
	calc9681: LREAL :=  10;
	calc9682: LREAL :=  10;
	calc9683: LREAL :=  10;
	calc9684: LREAL :=  10;
	calc9685: LREAL :=  10;
	calc9686: LREAL :=  10;
	calc9687: LREAL :=  10;
	calc9688: LREAL :=  10;
	calc9689: LREAL :=  10;
	calc9690: LREAL :=  10;
	calc9691: LREAL :=  10;
	calc9692: LREAL :=  10;
	calc9693: LREAL :=  10;
	calc9694: LREAL :=  10;
	calc9695: LREAL :=  10;
	calc9696: LREAL :=  10;
	calc9697: LREAL :=  10;
	calc9698: LREAL :=  10;
	calc9699: LREAL :=  10;
	calc9700: LREAL :=  10;
	calc9701: LREAL :=  10;
	calc9702: LREAL :=  10;
	calc9703: LREAL :=  10;
	calc9704: LREAL :=  10;
	calc9705: LREAL :=  10;
	calc9706: LREAL :=  10;
	calc9707: LREAL :=  10;
	calc9708: LREAL :=  10;
	calc9709: LREAL :=  10;
	calc9710: LREAL :=  10;
	calc9711: LREAL :=  10;
	calc9712: LREAL :=  10;
	calc9713: LREAL :=  10;
	calc9714: LREAL :=  10;
	calc9715: LREAL :=  10;
	calc9716: LREAL :=  10;
	calc9717: LREAL :=  10;
	calc9718: LREAL :=  10;
	calc9719: LREAL :=  10;
	calc9720: LREAL :=  10;
	calc9721: LREAL :=  10;
	calc9722: LREAL :=  10;
	calc9723: LREAL :=  10;
	calc9724: LREAL :=  10;
	calc9725: LREAL :=  10;
	calc9726: LREAL :=  10;
	calc9727: LREAL :=  10;
	calc9728: LREAL :=  10;
	calc9729: LREAL :=  10;
	calc9730: LREAL :=  10;
	calc9731: LREAL :=  10;
	calc9732: LREAL :=  10;
	calc9733: LREAL :=  10;
	calc9734: LREAL :=  10;
	calc9735: LREAL :=  10;
	calc9736: LREAL :=  10;
	calc9737: LREAL :=  10;
	calc9738: LREAL :=  10;
	calc9739: LREAL :=  10;
	calc9740: LREAL :=  10;
	calc9741: LREAL :=  10;
	calc9742: LREAL :=  10;
	calc9743: LREAL :=  10;
	calc9744: LREAL :=  10;
	calc9745: LREAL :=  10;
	calc9746: LREAL :=  10;
	calc9747: LREAL :=  10;
	calc9748: LREAL :=  10;
	calc9749: LREAL :=  10;
	calc9750: LREAL :=  10;
	calc9751: LREAL :=  10;
	calc9752: LREAL :=  10;
	calc9753: LREAL :=  10;
	calc9754: LREAL :=  10;
	calc9755: LREAL :=  10;
	calc9756: LREAL :=  10;
	calc9757: LREAL :=  10;
	calc9758: LREAL :=  10;
	calc9759: LREAL :=  10;
	calc9760: LREAL :=  10;
	calc9761: LREAL :=  10;
	calc9762: LREAL :=  10;
	calc9763: LREAL :=  10;
	calc9764: LREAL :=  10;
	calc9765: LREAL :=  10;
	calc9766: LREAL :=  10;
	calc9767: LREAL :=  10;
	calc9768: LREAL :=  10;
	calc9769: LREAL :=  10;
	calc9770: LREAL :=  10;
	calc9771: LREAL :=  10;
	calc9772: LREAL :=  10;
	calc9773: LREAL :=  10;
	calc9774: LREAL :=  10;
	calc9775: LREAL :=  10;
	calc9776: LREAL :=  10;
	calc9777: LREAL :=  10;
	calc9778: LREAL :=  10;
	calc9779: LREAL :=  10;
	calc9780: LREAL :=  10;
	calc9781: LREAL :=  10;
	calc9782: LREAL :=  10;
	calc9783: LREAL :=  10;
	calc9784: LREAL :=  10;
	calc9785: LREAL :=  10;
	calc9786: LREAL :=  10;
	calc9787: LREAL :=  10;
	calc9788: LREAL :=  10;
	calc9789: LREAL :=  10;
	calc9790: LREAL :=  10;
	calc9791: LREAL :=  10;
	calc9792: LREAL :=  10;
	calc9793: LREAL :=  10;
	calc9794: LREAL :=  10;
	calc9795: LREAL :=  10;
	calc9796: LREAL :=  10;
	calc9797: LREAL :=  10;
	calc9798: LREAL :=  10;
	calc9799: LREAL :=  10;
	calc9800: LREAL :=  10;
	calc9801: LREAL :=  10;
	calc9802: LREAL :=  10;
	calc9803: LREAL :=  10;
	calc9804: LREAL :=  10;
	calc9805: LREAL :=  10;
	calc9806: LREAL :=  10;
	calc9807: LREAL :=  10;
	calc9808: LREAL :=  10;
	calc9809: LREAL :=  10;
	calc9810: LREAL :=  10;
	calc9811: LREAL :=  10;
	calc9812: LREAL :=  10;
	calc9813: LREAL :=  10;
	calc9814: LREAL :=  10;
	calc9815: LREAL :=  10;
	calc9816: LREAL :=  10;
	calc9817: LREAL :=  10;
	calc9818: LREAL :=  10;
	calc9819: LREAL :=  10;
	calc9820: LREAL :=  10;
	calc9821: LREAL :=  10;
	calc9822: LREAL :=  10;
	calc9823: LREAL :=  10;
	calc9824: LREAL :=  10;
	calc9825: LREAL :=  10;
	calc9826: LREAL :=  10;
	calc9827: LREAL :=  10;
	calc9828: LREAL :=  10;
	calc9829: LREAL :=  10;
	calc9830: LREAL :=  10;
	calc9831: LREAL :=  10;
	calc9832: LREAL :=  10;
	calc9833: LREAL :=  10;
	calc9834: LREAL :=  10;
	calc9835: LREAL :=  10;
	calc9836: LREAL :=  10;
	calc9837: LREAL :=  10;
	calc9838: LREAL :=  10;
	calc9839: LREAL :=  10;
	calc9840: LREAL :=  10;
	calc9841: LREAL :=  10;
	calc9842: LREAL :=  10;
	calc9843: LREAL :=  10;
	calc9844: LREAL :=  10;
	calc9845: LREAL :=  10;
	calc9846: LREAL :=  10;
	calc9847: LREAL :=  10;
	calc9848: LREAL :=  10;
	calc9849: LREAL :=  10;
	calc9850: LREAL :=  10;
	calc9851: LREAL :=  10;
	calc9852: LREAL :=  10;
	calc9853: LREAL :=  10;
	calc9854: LREAL :=  10;
	calc9855: LREAL :=  10;
	calc9856: LREAL :=  10;
	calc9857: LREAL :=  10;
	calc9858: LREAL :=  10;
	calc9859: LREAL :=  10;
	calc9860: LREAL :=  10;
	calc9861: LREAL :=  10;
	calc9862: LREAL :=  10;
	calc9863: LREAL :=  10;
	calc9864: LREAL :=  10;
	calc9865: LREAL :=  10;
	calc9866: LREAL :=  10;
	calc9867: LREAL :=  10;
	calc9868: LREAL :=  10;
	calc9869: LREAL :=  10;
	calc9870: LREAL :=  10;
	calc9871: LREAL :=  10;
	calc9872: LREAL :=  10;
	calc9873: LREAL :=  10;
	calc9874: LREAL :=  10;
	calc9875: LREAL :=  10;
	calc9876: LREAL :=  10;
	calc9877: LREAL :=  10;
	calc9878: LREAL :=  10;
	calc9879: LREAL :=  10;
	calc9880: LREAL :=  10;
	calc9881: LREAL :=  10;
	calc9882: LREAL :=  10;
	calc9883: LREAL :=  10;
	calc9884: LREAL :=  10;
	calc9885: LREAL :=  10;
	calc9886: LREAL :=  10;
	calc9887: LREAL :=  10;
	calc9888: LREAL :=  10;
	calc9889: LREAL :=  10;
	calc9890: LREAL :=  10;
	calc9891: LREAL :=  10;
	calc9892: LREAL :=  10;
	calc9893: LREAL :=  10;
	calc9894: LREAL :=  10;
	calc9895: LREAL :=  10;
	calc9896: LREAL :=  10;
	calc9897: LREAL :=  10;
	calc9898: LREAL :=  10;
	calc9899: LREAL :=  10;
	calc9900: LREAL :=  10;
	calc9901: LREAL :=  10;
	calc9902: LREAL :=  10;
	calc9903: LREAL :=  10;
	calc9904: LREAL :=  10;
	calc9905: LREAL :=  10;
	calc9906: LREAL :=  10;
	calc9907: LREAL :=  10;
	calc9908: LREAL :=  10;
	calc9909: LREAL :=  10;
	calc9910: LREAL :=  10;
	calc9911: LREAL :=  10;
	calc9912: LREAL :=  10;
	calc9913: LREAL :=  10;
	calc9914: LREAL :=  10;
	calc9915: LREAL :=  10;
	calc9916: LREAL :=  10;
	calc9917: LREAL :=  10;
	calc9918: LREAL :=  10;
	calc9919: LREAL :=  10;
	calc9920: LREAL :=  10;
	calc9921: LREAL :=  10;
	calc9922: LREAL :=  10;
	calc9923: LREAL :=  10;
	calc9924: LREAL :=  10;
	calc9925: LREAL :=  10;
	calc9926: LREAL :=  10;
	calc9927: LREAL :=  10;
	calc9928: LREAL :=  10;
	calc9929: LREAL :=  10;
	calc9930: LREAL :=  10;
	calc9931: LREAL :=  10;
	calc9932: LREAL :=  10;
	calc9933: LREAL :=  10;
	calc9934: LREAL :=  10;
	calc9935: LREAL :=  10;
	calc9936: LREAL :=  10;
	calc9937: LREAL :=  10;
	calc9938: LREAL :=  10;
	calc9939: LREAL :=  10;
	calc9940: LREAL :=  10;
	calc9941: LREAL :=  10;
	calc9942: LREAL :=  10;
	calc9943: LREAL :=  10;
	calc9944: LREAL :=  10;
	calc9945: LREAL :=  10;
	calc9946: LREAL :=  10;
	calc9947: LREAL :=  10;
	calc9948: LREAL :=  10;
	calc9949: LREAL :=  10;
	calc9950: LREAL :=  10;
	calc9951: LREAL :=  10;
	calc9952: LREAL :=  10;
	calc9953: LREAL :=  10;
	calc9954: LREAL :=  10;
	calc9955: LREAL :=  10;
	calc9956: LREAL :=  10;
	calc9957: LREAL :=  10;
	calc9958: LREAL :=  10;
	calc9959: LREAL :=  10;
	calc9960: LREAL :=  10;
	calc9961: LREAL :=  10;
	calc9962: LREAL :=  10;
	calc9963: LREAL :=  10;
	calc9964: LREAL :=  10;
	calc9965: LREAL :=  10;
	calc9966: LREAL :=  10;
	calc9967: LREAL :=  10;
	calc9968: LREAL :=  10;
	calc9969: LREAL :=  10;
	calc9970: LREAL :=  10;
	calc9971: LREAL :=  10;
	calc9972: LREAL :=  10;
	calc9973: LREAL :=  10;
	calc9974: LREAL :=  10;
	calc9975: LREAL :=  10;
	calc9976: LREAL :=  10;
	calc9977: LREAL :=  10;
	calc9978: LREAL :=  10;
	calc9979: LREAL :=  10;
	calc9980: LREAL :=  10;
	calc9981: LREAL :=  10;
	calc9982: LREAL :=  10;
	calc9983: LREAL :=  10;
	calc9984: LREAL :=  10;
	calc9985: LREAL :=  10;
	calc9986: LREAL :=  10;
	calc9987: LREAL :=  10;
	calc9988: LREAL :=  10;
	calc9989: LREAL :=  10;
	calc9990: LREAL :=  10;
	calc9991: LREAL :=  10;
	calc9992: LREAL :=  10;
	calc9993: LREAL :=  10;
	calc9994: LREAL :=  10;
	calc9995: LREAL :=  10;
	calc9996: LREAL :=  10;
	calc9997: LREAL :=  10;
	calc9998: LREAL :=  10;
	calc9999: LREAL :=  10;
	
		counter0: LREAL :=  0;
	counter1: LREAL :=  0;
	counter2: LREAL :=  0;
	counter3: LREAL :=  0;
	counter4: LREAL :=  0;
	counter5: LREAL :=  0;
	counter6: LREAL :=  0;
	counter7: LREAL :=  0;
	counter8: LREAL :=  0;
	counter9: LREAL :=  0;
	counter10: LREAL :=  0;
	counter11: LREAL :=  0;
	counter12: LREAL :=  0;
	counter13: LREAL :=  0;
	counter14: LREAL :=  0;
	counter15: LREAL :=  0;
	counter16: LREAL :=  0;
	counter17: LREAL :=  0;
	counter18: LREAL :=  0;
	counter19: LREAL :=  0;
	counter20: LREAL :=  0;
	counter21: LREAL :=  0;
	counter22: LREAL :=  0;
	counter23: LREAL :=  0;
	counter24: LREAL :=  0;
	counter25: LREAL :=  0;
	counter26: LREAL :=  0;
	counter27: LREAL :=  0;
	counter28: LREAL :=  0;
	counter29: LREAL :=  0;
	counter30: LREAL :=  0;
	counter31: LREAL :=  0;
	counter32: LREAL :=  0;
	counter33: LREAL :=  0;
	counter34: LREAL :=  0;
	counter35: LREAL :=  0;
	counter36: LREAL :=  0;
	counter37: LREAL :=  0;
	counter38: LREAL :=  0;
	counter39: LREAL :=  0;
	counter40: LREAL :=  0;
	counter41: LREAL :=  0;
	counter42: LREAL :=  0;
	counter43: LREAL :=  0;
	counter44: LREAL :=  0;
	counter45: LREAL :=  0;
	counter46: LREAL :=  0;
	counter47: LREAL :=  0;
	counter48: LREAL :=  0;
	counter49: LREAL :=  0;
	counter50: LREAL :=  0;
	counter51: LREAL :=  0;
	counter52: LREAL :=  0;
	counter53: LREAL :=  0;
	counter54: LREAL :=  0;
	counter55: LREAL :=  0;
	counter56: LREAL :=  0;
	counter57: LREAL :=  0;
	counter58: LREAL :=  0;
	counter59: LREAL :=  0;
	counter60: LREAL :=  0;
	counter61: LREAL :=  0;
	counter62: LREAL :=  0;
	counter63: LREAL :=  0;
	counter64: LREAL :=  0;
	counter65: LREAL :=  0;
	counter66: LREAL :=  0;
	counter67: LREAL :=  0;
	counter68: LREAL :=  0;
	counter69: LREAL :=  0;
	counter70: LREAL :=  0;
	counter71: LREAL :=  0;
	counter72: LREAL :=  0;
	counter73: LREAL :=  0;
	counter74: LREAL :=  0;
	counter75: LREAL :=  0;
	counter76: LREAL :=  0;
	counter77: LREAL :=  0;
	counter78: LREAL :=  0;
	counter79: LREAL :=  0;
	counter80: LREAL :=  0;
	counter81: LREAL :=  0;
	counter82: LREAL :=  0;
	counter83: LREAL :=  0;
	counter84: LREAL :=  0;
	counter85: LREAL :=  0;
	counter86: LREAL :=  0;
	counter87: LREAL :=  0;
	counter88: LREAL :=  0;
	counter89: LREAL :=  0;
	counter90: LREAL :=  0;
	counter91: LREAL :=  0;
	counter92: LREAL :=  0;
	counter93: LREAL :=  0;
	counter94: LREAL :=  0;
	counter95: LREAL :=  0;
	counter96: LREAL :=  0;
	counter97: LREAL :=  0;
	counter98: LREAL :=  0;
	counter99: LREAL :=  0;
	counter100: LREAL :=  0;
	counter101: LREAL :=  0;
	counter102: LREAL :=  0;
	counter103: LREAL :=  0;
	counter104: LREAL :=  0;
	counter105: LREAL :=  0;
	counter106: LREAL :=  0;
	counter107: LREAL :=  0;
	counter108: LREAL :=  0;
	counter109: LREAL :=  0;
	counter110: LREAL :=  0;
	counter111: LREAL :=  0;
	counter112: LREAL :=  0;
	counter113: LREAL :=  0;
	counter114: LREAL :=  0;
	counter115: LREAL :=  0;
	counter116: LREAL :=  0;
	counter117: LREAL :=  0;
	counter118: LREAL :=  0;
	counter119: LREAL :=  0;
	counter120: LREAL :=  0;
	counter121: LREAL :=  0;
	counter122: LREAL :=  0;
	counter123: LREAL :=  0;
	counter124: LREAL :=  0;
	counter125: LREAL :=  0;
	counter126: LREAL :=  0;
	counter127: LREAL :=  0;
	counter128: LREAL :=  0;
	counter129: LREAL :=  0;
	counter130: LREAL :=  0;
	counter131: LREAL :=  0;
	counter132: LREAL :=  0;
	counter133: LREAL :=  0;
	counter134: LREAL :=  0;
	counter135: LREAL :=  0;
	counter136: LREAL :=  0;
	counter137: LREAL :=  0;
	counter138: LREAL :=  0;
	counter139: LREAL :=  0;
	counter140: LREAL :=  0;
	counter141: LREAL :=  0;
	counter142: LREAL :=  0;
	counter143: LREAL :=  0;
	counter144: LREAL :=  0;
	counter145: LREAL :=  0;
	counter146: LREAL :=  0;
	counter147: LREAL :=  0;
	counter148: LREAL :=  0;
	counter149: LREAL :=  0;
	counter150: LREAL :=  0;
	counter151: LREAL :=  0;
	counter152: LREAL :=  0;
	counter153: LREAL :=  0;
	counter154: LREAL :=  0;
	counter155: LREAL :=  0;
	counter156: LREAL :=  0;
	counter157: LREAL :=  0;
	counter158: LREAL :=  0;
	counter159: LREAL :=  0;
	counter160: LREAL :=  0;
	counter161: LREAL :=  0;
	counter162: LREAL :=  0;
	counter163: LREAL :=  0;
	counter164: LREAL :=  0;
	counter165: LREAL :=  0;
	counter166: LREAL :=  0;
	counter167: LREAL :=  0;
	counter168: LREAL :=  0;
	counter169: LREAL :=  0;
	counter170: LREAL :=  0;
	counter171: LREAL :=  0;
	counter172: LREAL :=  0;
	counter173: LREAL :=  0;
	counter174: LREAL :=  0;
	counter175: LREAL :=  0;
	counter176: LREAL :=  0;
	counter177: LREAL :=  0;
	counter178: LREAL :=  0;
	counter179: LREAL :=  0;
	counter180: LREAL :=  0;
	counter181: LREAL :=  0;
	counter182: LREAL :=  0;
	counter183: LREAL :=  0;
	counter184: LREAL :=  0;
	counter185: LREAL :=  0;
	counter186: LREAL :=  0;
	counter187: LREAL :=  0;
	counter188: LREAL :=  0;
	counter189: LREAL :=  0;
	counter190: LREAL :=  0;
	counter191: LREAL :=  0;
	counter192: LREAL :=  0;
	counter193: LREAL :=  0;
	counter194: LREAL :=  0;
	counter195: LREAL :=  0;
	counter196: LREAL :=  0;
	counter197: LREAL :=  0;
	counter198: LREAL :=  0;
	counter199: LREAL :=  0;
	counter200: LREAL :=  0;
	counter201: LREAL :=  0;
	counter202: LREAL :=  0;
	counter203: LREAL :=  0;
	counter204: LREAL :=  0;
	counter205: LREAL :=  0;
	counter206: LREAL :=  0;
	counter207: LREAL :=  0;
	counter208: LREAL :=  0;
	counter209: LREAL :=  0;
	counter210: LREAL :=  0;
	counter211: LREAL :=  0;
	counter212: LREAL :=  0;
	counter213: LREAL :=  0;
	counter214: LREAL :=  0;
	counter215: LREAL :=  0;
	counter216: LREAL :=  0;
	counter217: LREAL :=  0;
	counter218: LREAL :=  0;
	counter219: LREAL :=  0;
	counter220: LREAL :=  0;
	counter221: LREAL :=  0;
	counter222: LREAL :=  0;
	counter223: LREAL :=  0;
	counter224: LREAL :=  0;
	counter225: LREAL :=  0;
	counter226: LREAL :=  0;
	counter227: LREAL :=  0;
	counter228: LREAL :=  0;
	counter229: LREAL :=  0;
	counter230: LREAL :=  0;
	counter231: LREAL :=  0;
	counter232: LREAL :=  0;
	counter233: LREAL :=  0;
	counter234: LREAL :=  0;
	counter235: LREAL :=  0;
	counter236: LREAL :=  0;
	counter237: LREAL :=  0;
	counter238: LREAL :=  0;
	counter239: LREAL :=  0;
	counter240: LREAL :=  0;
	counter241: LREAL :=  0;
	counter242: LREAL :=  0;
	counter243: LREAL :=  0;
	counter244: LREAL :=  0;
	counter245: LREAL :=  0;
	counter246: LREAL :=  0;
	counter247: LREAL :=  0;
	counter248: LREAL :=  0;
	counter249: LREAL :=  0;
	counter250: LREAL :=  0;
	counter251: LREAL :=  0;
	counter252: LREAL :=  0;
	counter253: LREAL :=  0;
	counter254: LREAL :=  0;
	counter255: LREAL :=  0;
	counter256: LREAL :=  0;
	counter257: LREAL :=  0;
	counter258: LREAL :=  0;
	counter259: LREAL :=  0;
	counter260: LREAL :=  0;
	counter261: LREAL :=  0;
	counter262: LREAL :=  0;
	counter263: LREAL :=  0;
	counter264: LREAL :=  0;
	counter265: LREAL :=  0;
	counter266: LREAL :=  0;
	counter267: LREAL :=  0;
	counter268: LREAL :=  0;
	counter269: LREAL :=  0;
	counter270: LREAL :=  0;
	counter271: LREAL :=  0;
	counter272: LREAL :=  0;
	counter273: LREAL :=  0;
	counter274: LREAL :=  0;
	counter275: LREAL :=  0;
	counter276: LREAL :=  0;
	counter277: LREAL :=  0;
	counter278: LREAL :=  0;
	counter279: LREAL :=  0;
	counter280: LREAL :=  0;
	counter281: LREAL :=  0;
	counter282: LREAL :=  0;
	counter283: LREAL :=  0;
	counter284: LREAL :=  0;
	counter285: LREAL :=  0;
	counter286: LREAL :=  0;
	counter287: LREAL :=  0;
	counter288: LREAL :=  0;
	counter289: LREAL :=  0;
	counter290: LREAL :=  0;
	counter291: LREAL :=  0;
	counter292: LREAL :=  0;
	counter293: LREAL :=  0;
	counter294: LREAL :=  0;
	counter295: LREAL :=  0;
	counter296: LREAL :=  0;
	counter297: LREAL :=  0;
	counter298: LREAL :=  0;
	counter299: LREAL :=  0;
	counter300: LREAL :=  0;
	counter301: LREAL :=  0;
	counter302: LREAL :=  0;
	counter303: LREAL :=  0;
	counter304: LREAL :=  0;
	counter305: LREAL :=  0;
	counter306: LREAL :=  0;
	counter307: LREAL :=  0;
	counter308: LREAL :=  0;
	counter309: LREAL :=  0;
	counter310: LREAL :=  0;
	counter311: LREAL :=  0;
	counter312: LREAL :=  0;
	counter313: LREAL :=  0;
	counter314: LREAL :=  0;
	counter315: LREAL :=  0;
	counter316: LREAL :=  0;
	counter317: LREAL :=  0;
	counter318: LREAL :=  0;
	counter319: LREAL :=  0;
	counter320: LREAL :=  0;
	counter321: LREAL :=  0;
	counter322: LREAL :=  0;
	counter323: LREAL :=  0;
	counter324: LREAL :=  0;
	counter325: LREAL :=  0;
	counter326: LREAL :=  0;
	counter327: LREAL :=  0;
	counter328: LREAL :=  0;
	counter329: LREAL :=  0;
	counter330: LREAL :=  0;
	counter331: LREAL :=  0;
	counter332: LREAL :=  0;
	counter333: LREAL :=  0;
	counter334: LREAL :=  0;
	counter335: LREAL :=  0;
	counter336: LREAL :=  0;
	counter337: LREAL :=  0;
	counter338: LREAL :=  0;
	counter339: LREAL :=  0;
	counter340: LREAL :=  0;
	counter341: LREAL :=  0;
	counter342: LREAL :=  0;
	counter343: LREAL :=  0;
	counter344: LREAL :=  0;
	counter345: LREAL :=  0;
	counter346: LREAL :=  0;
	counter347: LREAL :=  0;
	counter348: LREAL :=  0;
	counter349: LREAL :=  0;
	counter350: LREAL :=  0;
	counter351: LREAL :=  0;
	counter352: LREAL :=  0;
	counter353: LREAL :=  0;
	counter354: LREAL :=  0;
	counter355: LREAL :=  0;
	counter356: LREAL :=  0;
	counter357: LREAL :=  0;
	counter358: LREAL :=  0;
	counter359: LREAL :=  0;
	counter360: LREAL :=  0;
	counter361: LREAL :=  0;
	counter362: LREAL :=  0;
	counter363: LREAL :=  0;
	counter364: LREAL :=  0;
	counter365: LREAL :=  0;
	counter366: LREAL :=  0;
	counter367: LREAL :=  0;
	counter368: LREAL :=  0;
	counter369: LREAL :=  0;
	counter370: LREAL :=  0;
	counter371: LREAL :=  0;
	counter372: LREAL :=  0;
	counter373: LREAL :=  0;
	counter374: LREAL :=  0;
	counter375: LREAL :=  0;
	counter376: LREAL :=  0;
	counter377: LREAL :=  0;
	counter378: LREAL :=  0;
	counter379: LREAL :=  0;
	counter380: LREAL :=  0;
	counter381: LREAL :=  0;
	counter382: LREAL :=  0;
	counter383: LREAL :=  0;
	counter384: LREAL :=  0;
	counter385: LREAL :=  0;
	counter386: LREAL :=  0;
	counter387: LREAL :=  0;
	counter388: LREAL :=  0;
	counter389: LREAL :=  0;
	counter390: LREAL :=  0;
	counter391: LREAL :=  0;
	counter392: LREAL :=  0;
	counter393: LREAL :=  0;
	counter394: LREAL :=  0;
	counter395: LREAL :=  0;
	counter396: LREAL :=  0;
	counter397: LREAL :=  0;
	counter398: LREAL :=  0;
	counter399: LREAL :=  0;
	counter400: LREAL :=  0;
	counter401: LREAL :=  0;
	counter402: LREAL :=  0;
	counter403: LREAL :=  0;
	counter404: LREAL :=  0;
	counter405: LREAL :=  0;
	counter406: LREAL :=  0;
	counter407: LREAL :=  0;
	counter408: LREAL :=  0;
	counter409: LREAL :=  0;
	counter410: LREAL :=  0;
	counter411: LREAL :=  0;
	counter412: LREAL :=  0;
	counter413: LREAL :=  0;
	counter414: LREAL :=  0;
	counter415: LREAL :=  0;
	counter416: LREAL :=  0;
	counter417: LREAL :=  0;
	counter418: LREAL :=  0;
	counter419: LREAL :=  0;
	counter420: LREAL :=  0;
	counter421: LREAL :=  0;
	counter422: LREAL :=  0;
	counter423: LREAL :=  0;
	counter424: LREAL :=  0;
	counter425: LREAL :=  0;
	counter426: LREAL :=  0;
	counter427: LREAL :=  0;
	counter428: LREAL :=  0;
	counter429: LREAL :=  0;
	counter430: LREAL :=  0;
	counter431: LREAL :=  0;
	counter432: LREAL :=  0;
	counter433: LREAL :=  0;
	counter434: LREAL :=  0;
	counter435: LREAL :=  0;
	counter436: LREAL :=  0;
	counter437: LREAL :=  0;
	counter438: LREAL :=  0;
	counter439: LREAL :=  0;
	counter440: LREAL :=  0;
	counter441: LREAL :=  0;
	counter442: LREAL :=  0;
	counter443: LREAL :=  0;
	counter444: LREAL :=  0;
	counter445: LREAL :=  0;
	counter446: LREAL :=  0;
	counter447: LREAL :=  0;
	counter448: LREAL :=  0;
	counter449: LREAL :=  0;
	counter450: LREAL :=  0;
	counter451: LREAL :=  0;
	counter452: LREAL :=  0;
	counter453: LREAL :=  0;
	counter454: LREAL :=  0;
	counter455: LREAL :=  0;
	counter456: LREAL :=  0;
	counter457: LREAL :=  0;
	counter458: LREAL :=  0;
	counter459: LREAL :=  0;
	counter460: LREAL :=  0;
	counter461: LREAL :=  0;
	counter462: LREAL :=  0;
	counter463: LREAL :=  0;
	counter464: LREAL :=  0;
	counter465: LREAL :=  0;
	counter466: LREAL :=  0;
	counter467: LREAL :=  0;
	counter468: LREAL :=  0;
	counter469: LREAL :=  0;
	counter470: LREAL :=  0;
	counter471: LREAL :=  0;
	counter472: LREAL :=  0;
	counter473: LREAL :=  0;
	counter474: LREAL :=  0;
	counter475: LREAL :=  0;
	counter476: LREAL :=  0;
	counter477: LREAL :=  0;
	counter478: LREAL :=  0;
	counter479: LREAL :=  0;
	counter480: LREAL :=  0;
	counter481: LREAL :=  0;
	counter482: LREAL :=  0;
	counter483: LREAL :=  0;
	counter484: LREAL :=  0;
	counter485: LREAL :=  0;
	counter486: LREAL :=  0;
	counter487: LREAL :=  0;
	counter488: LREAL :=  0;
	counter489: LREAL :=  0;
	counter490: LREAL :=  0;
	counter491: LREAL :=  0;
	counter492: LREAL :=  0;
	counter493: LREAL :=  0;
	counter494: LREAL :=  0;
	counter495: LREAL :=  0;
	counter496: LREAL :=  0;
	counter497: LREAL :=  0;
	counter498: LREAL :=  0;
	counter499: LREAL :=  0;
	counter500: LREAL :=  0;
	counter501: LREAL :=  0;
	counter502: LREAL :=  0;
	counter503: LREAL :=  0;
	counter504: LREAL :=  0;
	counter505: LREAL :=  0;
	counter506: LREAL :=  0;
	counter507: LREAL :=  0;
	counter508: LREAL :=  0;
	counter509: LREAL :=  0;
	counter510: LREAL :=  0;
	counter511: LREAL :=  0;
	counter512: LREAL :=  0;
	counter513: LREAL :=  0;
	counter514: LREAL :=  0;
	counter515: LREAL :=  0;
	counter516: LREAL :=  0;
	counter517: LREAL :=  0;
	counter518: LREAL :=  0;
	counter519: LREAL :=  0;
	counter520: LREAL :=  0;
	counter521: LREAL :=  0;
	counter522: LREAL :=  0;
	counter523: LREAL :=  0;
	counter524: LREAL :=  0;
	counter525: LREAL :=  0;
	counter526: LREAL :=  0;
	counter527: LREAL :=  0;
	counter528: LREAL :=  0;
	counter529: LREAL :=  0;
	counter530: LREAL :=  0;
	counter531: LREAL :=  0;
	counter532: LREAL :=  0;
	counter533: LREAL :=  0;
	counter534: LREAL :=  0;
	counter535: LREAL :=  0;
	counter536: LREAL :=  0;
	counter537: LREAL :=  0;
	counter538: LREAL :=  0;
	counter539: LREAL :=  0;
	counter540: LREAL :=  0;
	counter541: LREAL :=  0;
	counter542: LREAL :=  0;
	counter543: LREAL :=  0;
	counter544: LREAL :=  0;
	counter545: LREAL :=  0;
	counter546: LREAL :=  0;
	counter547: LREAL :=  0;
	counter548: LREAL :=  0;
	counter549: LREAL :=  0;
	counter550: LREAL :=  0;
	counter551: LREAL :=  0;
	counter552: LREAL :=  0;
	counter553: LREAL :=  0;
	counter554: LREAL :=  0;
	counter555: LREAL :=  0;
	counter556: LREAL :=  0;
	counter557: LREAL :=  0;
	counter558: LREAL :=  0;
	counter559: LREAL :=  0;
	counter560: LREAL :=  0;
	counter561: LREAL :=  0;
	counter562: LREAL :=  0;
	counter563: LREAL :=  0;
	counter564: LREAL :=  0;
	counter565: LREAL :=  0;
	counter566: LREAL :=  0;
	counter567: LREAL :=  0;
	counter568: LREAL :=  0;
	counter569: LREAL :=  0;
	counter570: LREAL :=  0;
	counter571: LREAL :=  0;
	counter572: LREAL :=  0;
	counter573: LREAL :=  0;
	counter574: LREAL :=  0;
	counter575: LREAL :=  0;
	counter576: LREAL :=  0;
	counter577: LREAL :=  0;
	counter578: LREAL :=  0;
	counter579: LREAL :=  0;
	counter580: LREAL :=  0;
	counter581: LREAL :=  0;
	counter582: LREAL :=  0;
	counter583: LREAL :=  0;
	counter584: LREAL :=  0;
	counter585: LREAL :=  0;
	counter586: LREAL :=  0;
	counter587: LREAL :=  0;
	counter588: LREAL :=  0;
	counter589: LREAL :=  0;
	counter590: LREAL :=  0;
	counter591: LREAL :=  0;
	counter592: LREAL :=  0;
	counter593: LREAL :=  0;
	counter594: LREAL :=  0;
	counter595: LREAL :=  0;
	counter596: LREAL :=  0;
	counter597: LREAL :=  0;
	counter598: LREAL :=  0;
	counter599: LREAL :=  0;
	counter600: LREAL :=  0;
	counter601: LREAL :=  0;
	counter602: LREAL :=  0;
	counter603: LREAL :=  0;
	counter604: LREAL :=  0;
	counter605: LREAL :=  0;
	counter606: LREAL :=  0;
	counter607: LREAL :=  0;
	counter608: LREAL :=  0;
	counter609: LREAL :=  0;
	counter610: LREAL :=  0;
	counter611: LREAL :=  0;
	counter612: LREAL :=  0;
	counter613: LREAL :=  0;
	counter614: LREAL :=  0;
	counter615: LREAL :=  0;
	counter616: LREAL :=  0;
	counter617: LREAL :=  0;
	counter618: LREAL :=  0;
	counter619: LREAL :=  0;
	counter620: LREAL :=  0;
	counter621: LREAL :=  0;
	counter622: LREAL :=  0;
	counter623: LREAL :=  0;
	counter624: LREAL :=  0;
	counter625: LREAL :=  0;
	counter626: LREAL :=  0;
	counter627: LREAL :=  0;
	counter628: LREAL :=  0;
	counter629: LREAL :=  0;
	counter630: LREAL :=  0;
	counter631: LREAL :=  0;
	counter632: LREAL :=  0;
	counter633: LREAL :=  0;
	counter634: LREAL :=  0;
	counter635: LREAL :=  0;
	counter636: LREAL :=  0;
	counter637: LREAL :=  0;
	counter638: LREAL :=  0;
	counter639: LREAL :=  0;
	counter640: LREAL :=  0;
	counter641: LREAL :=  0;
	counter642: LREAL :=  0;
	counter643: LREAL :=  0;
	counter644: LREAL :=  0;
	counter645: LREAL :=  0;
	counter646: LREAL :=  0;
	counter647: LREAL :=  0;
	counter648: LREAL :=  0;
	counter649: LREAL :=  0;
	counter650: LREAL :=  0;
	counter651: LREAL :=  0;
	counter652: LREAL :=  0;
	counter653: LREAL :=  0;
	counter654: LREAL :=  0;
	counter655: LREAL :=  0;
	counter656: LREAL :=  0;
	counter657: LREAL :=  0;
	counter658: LREAL :=  0;
	counter659: LREAL :=  0;
	counter660: LREAL :=  0;
	counter661: LREAL :=  0;
	counter662: LREAL :=  0;
	counter663: LREAL :=  0;
	counter664: LREAL :=  0;
	counter665: LREAL :=  0;
	counter666: LREAL :=  0;
	counter667: LREAL :=  0;
	counter668: LREAL :=  0;
	counter669: LREAL :=  0;
	counter670: LREAL :=  0;
	counter671: LREAL :=  0;
	counter672: LREAL :=  0;
	counter673: LREAL :=  0;
	counter674: LREAL :=  0;
	counter675: LREAL :=  0;
	counter676: LREAL :=  0;
	counter677: LREAL :=  0;
	counter678: LREAL :=  0;
	counter679: LREAL :=  0;
	counter680: LREAL :=  0;
	counter681: LREAL :=  0;
	counter682: LREAL :=  0;
	counter683: LREAL :=  0;
	counter684: LREAL :=  0;
	counter685: LREAL :=  0;
	counter686: LREAL :=  0;
	counter687: LREAL :=  0;
	counter688: LREAL :=  0;
	counter689: LREAL :=  0;
	counter690: LREAL :=  0;
	counter691: LREAL :=  0;
	counter692: LREAL :=  0;
	counter693: LREAL :=  0;
	counter694: LREAL :=  0;
	counter695: LREAL :=  0;
	counter696: LREAL :=  0;
	counter697: LREAL :=  0;
	counter698: LREAL :=  0;
	counter699: LREAL :=  0;
	counter700: LREAL :=  0;
	counter701: LREAL :=  0;
	counter702: LREAL :=  0;
	counter703: LREAL :=  0;
	counter704: LREAL :=  0;
	counter705: LREAL :=  0;
	counter706: LREAL :=  0;
	counter707: LREAL :=  0;
	counter708: LREAL :=  0;
	counter709: LREAL :=  0;
	counter710: LREAL :=  0;
	counter711: LREAL :=  0;
	counter712: LREAL :=  0;
	counter713: LREAL :=  0;
	counter714: LREAL :=  0;
	counter715: LREAL :=  0;
	counter716: LREAL :=  0;
	counter717: LREAL :=  0;
	counter718: LREAL :=  0;
	counter719: LREAL :=  0;
	counter720: LREAL :=  0;
	counter721: LREAL :=  0;
	counter722: LREAL :=  0;
	counter723: LREAL :=  0;
	counter724: LREAL :=  0;
	counter725: LREAL :=  0;
	counter726: LREAL :=  0;
	counter727: LREAL :=  0;
	counter728: LREAL :=  0;
	counter729: LREAL :=  0;
	counter730: LREAL :=  0;
	counter731: LREAL :=  0;
	counter732: LREAL :=  0;
	counter733: LREAL :=  0;
	counter734: LREAL :=  0;
	counter735: LREAL :=  0;
	counter736: LREAL :=  0;
	counter737: LREAL :=  0;
	counter738: LREAL :=  0;
	counter739: LREAL :=  0;
	counter740: LREAL :=  0;
	counter741: LREAL :=  0;
	counter742: LREAL :=  0;
	counter743: LREAL :=  0;
	counter744: LREAL :=  0;
	counter745: LREAL :=  0;
	counter746: LREAL :=  0;
	counter747: LREAL :=  0;
	counter748: LREAL :=  0;
	counter749: LREAL :=  0;
	counter750: LREAL :=  0;
	counter751: LREAL :=  0;
	counter752: LREAL :=  0;
	counter753: LREAL :=  0;
	counter754: LREAL :=  0;
	counter755: LREAL :=  0;
	counter756: LREAL :=  0;
	counter757: LREAL :=  0;
	counter758: LREAL :=  0;
	counter759: LREAL :=  0;
	counter760: LREAL :=  0;
	counter761: LREAL :=  0;
	counter762: LREAL :=  0;
	counter763: LREAL :=  0;
	counter764: LREAL :=  0;
	counter765: LREAL :=  0;
	counter766: LREAL :=  0;
	counter767: LREAL :=  0;
	counter768: LREAL :=  0;
	counter769: LREAL :=  0;
	counter770: LREAL :=  0;
	counter771: LREAL :=  0;
	counter772: LREAL :=  0;
	counter773: LREAL :=  0;
	counter774: LREAL :=  0;
	counter775: LREAL :=  0;
	counter776: LREAL :=  0;
	counter777: LREAL :=  0;
	counter778: LREAL :=  0;
	counter779: LREAL :=  0;
	counter780: LREAL :=  0;
	counter781: LREAL :=  0;
	counter782: LREAL :=  0;
	counter783: LREAL :=  0;
	counter784: LREAL :=  0;
	counter785: LREAL :=  0;
	counter786: LREAL :=  0;
	counter787: LREAL :=  0;
	counter788: LREAL :=  0;
	counter789: LREAL :=  0;
	counter790: LREAL :=  0;
	counter791: LREAL :=  0;
	counter792: LREAL :=  0;
	counter793: LREAL :=  0;
	counter794: LREAL :=  0;
	counter795: LREAL :=  0;
	counter796: LREAL :=  0;
	counter797: LREAL :=  0;
	counter798: LREAL :=  0;
	counter799: LREAL :=  0;
	counter800: LREAL :=  0;
	counter801: LREAL :=  0;
	counter802: LREAL :=  0;
	counter803: LREAL :=  0;
	counter804: LREAL :=  0;
	counter805: LREAL :=  0;
	counter806: LREAL :=  0;
	counter807: LREAL :=  0;
	counter808: LREAL :=  0;
	counter809: LREAL :=  0;
	counter810: LREAL :=  0;
	counter811: LREAL :=  0;
	counter812: LREAL :=  0;
	counter813: LREAL :=  0;
	counter814: LREAL :=  0;
	counter815: LREAL :=  0;
	counter816: LREAL :=  0;
	counter817: LREAL :=  0;
	counter818: LREAL :=  0;
	counter819: LREAL :=  0;
	counter820: LREAL :=  0;
	counter821: LREAL :=  0;
	counter822: LREAL :=  0;
	counter823: LREAL :=  0;
	counter824: LREAL :=  0;
	counter825: LREAL :=  0;
	counter826: LREAL :=  0;
	counter827: LREAL :=  0;
	counter828: LREAL :=  0;
	counter829: LREAL :=  0;
	counter830: LREAL :=  0;
	counter831: LREAL :=  0;
	counter832: LREAL :=  0;
	counter833: LREAL :=  0;
	counter834: LREAL :=  0;
	counter835: LREAL :=  0;
	counter836: LREAL :=  0;
	counter837: LREAL :=  0;
	counter838: LREAL :=  0;
	counter839: LREAL :=  0;
	counter840: LREAL :=  0;
	counter841: LREAL :=  0;
	counter842: LREAL :=  0;
	counter843: LREAL :=  0;
	counter844: LREAL :=  0;
	counter845: LREAL :=  0;
	counter846: LREAL :=  0;
	counter847: LREAL :=  0;
	counter848: LREAL :=  0;
	counter849: LREAL :=  0;
	counter850: LREAL :=  0;
	counter851: LREAL :=  0;
	counter852: LREAL :=  0;
	counter853: LREAL :=  0;
	counter854: LREAL :=  0;
	counter855: LREAL :=  0;
	counter856: LREAL :=  0;
	counter857: LREAL :=  0;
	counter858: LREAL :=  0;
	counter859: LREAL :=  0;
	counter860: LREAL :=  0;
	counter861: LREAL :=  0;
	counter862: LREAL :=  0;
	counter863: LREAL :=  0;
	counter864: LREAL :=  0;
	counter865: LREAL :=  0;
	counter866: LREAL :=  0;
	counter867: LREAL :=  0;
	counter868: LREAL :=  0;
	counter869: LREAL :=  0;
	counter870: LREAL :=  0;
	counter871: LREAL :=  0;
	counter872: LREAL :=  0;
	counter873: LREAL :=  0;
	counter874: LREAL :=  0;
	counter875: LREAL :=  0;
	counter876: LREAL :=  0;
	counter877: LREAL :=  0;
	counter878: LREAL :=  0;
	counter879: LREAL :=  0;
	counter880: LREAL :=  0;
	counter881: LREAL :=  0;
	counter882: LREAL :=  0;
	counter883: LREAL :=  0;
	counter884: LREAL :=  0;
	counter885: LREAL :=  0;
	counter886: LREAL :=  0;
	counter887: LREAL :=  0;
	counter888: LREAL :=  0;
	counter889: LREAL :=  0;
	counter890: LREAL :=  0;
	counter891: LREAL :=  0;
	counter892: LREAL :=  0;
	counter893: LREAL :=  0;
	counter894: LREAL :=  0;
	counter895: LREAL :=  0;
	counter896: LREAL :=  0;
	counter897: LREAL :=  0;
	counter898: LREAL :=  0;
	counter899: LREAL :=  0;
	counter900: LREAL :=  0;
	counter901: LREAL :=  0;
	counter902: LREAL :=  0;
	counter903: LREAL :=  0;
	counter904: LREAL :=  0;
	counter905: LREAL :=  0;
	counter906: LREAL :=  0;
	counter907: LREAL :=  0;
	counter908: LREAL :=  0;
	counter909: LREAL :=  0;
	counter910: LREAL :=  0;
	counter911: LREAL :=  0;
	counter912: LREAL :=  0;
	counter913: LREAL :=  0;
	counter914: LREAL :=  0;
	counter915: LREAL :=  0;
	counter916: LREAL :=  0;
	counter917: LREAL :=  0;
	counter918: LREAL :=  0;
	counter919: LREAL :=  0;
	counter920: LREAL :=  0;
	counter921: LREAL :=  0;
	counter922: LREAL :=  0;
	counter923: LREAL :=  0;
	counter924: LREAL :=  0;
	counter925: LREAL :=  0;
	counter926: LREAL :=  0;
	counter927: LREAL :=  0;
	counter928: LREAL :=  0;
	counter929: LREAL :=  0;
	counter930: LREAL :=  0;
	counter931: LREAL :=  0;
	counter932: LREAL :=  0;
	counter933: LREAL :=  0;
	counter934: LREAL :=  0;
	counter935: LREAL :=  0;
	counter936: LREAL :=  0;
	counter937: LREAL :=  0;
	counter938: LREAL :=  0;
	counter939: LREAL :=  0;
	counter940: LREAL :=  0;
	counter941: LREAL :=  0;
	counter942: LREAL :=  0;
	counter943: LREAL :=  0;
	counter944: LREAL :=  0;
	counter945: LREAL :=  0;
	counter946: LREAL :=  0;
	counter947: LREAL :=  0;
	counter948: LREAL :=  0;
	counter949: LREAL :=  0;
	counter950: LREAL :=  0;
	counter951: LREAL :=  0;
	counter952: LREAL :=  0;
	counter953: LREAL :=  0;
	counter954: LREAL :=  0;
	counter955: LREAL :=  0;
	counter956: LREAL :=  0;
	counter957: LREAL :=  0;
	counter958: LREAL :=  0;
	counter959: LREAL :=  0;
	counter960: LREAL :=  0;
	counter961: LREAL :=  0;
	counter962: LREAL :=  0;
	counter963: LREAL :=  0;
	counter964: LREAL :=  0;
	counter965: LREAL :=  0;
	counter966: LREAL :=  0;
	counter967: LREAL :=  0;
	counter968: LREAL :=  0;
	counter969: LREAL :=  0;
	counter970: LREAL :=  0;
	counter971: LREAL :=  0;
	counter972: LREAL :=  0;
	counter973: LREAL :=  0;
	counter974: LREAL :=  0;
	counter975: LREAL :=  0;
	counter976: LREAL :=  0;
	counter977: LREAL :=  0;
	counter978: LREAL :=  0;
	counter979: LREAL :=  0;
	counter980: LREAL :=  0;
	counter981: LREAL :=  0;
	counter982: LREAL :=  0;
	counter983: LREAL :=  0;
	counter984: LREAL :=  0;
	counter985: LREAL :=  0;
	counter986: LREAL :=  0;
	counter987: LREAL :=  0;
	counter988: LREAL :=  0;
	counter989: LREAL :=  0;
	counter990: LREAL :=  0;
	counter991: LREAL :=  0;
	counter992: LREAL :=  0;
	counter993: LREAL :=  0;
	counter994: LREAL :=  0;
	counter995: LREAL :=  0;
	counter996: LREAL :=  0;
	counter997: LREAL :=  0;
	counter998: LREAL :=  0;
	counter999: LREAL :=  0;
	counter1000: LREAL :=  0;
	counter1001: LREAL :=  0;
	counter1002: LREAL :=  0;
	counter1003: LREAL :=  0;
	counter1004: LREAL :=  0;
	counter1005: LREAL :=  0;
	counter1006: LREAL :=  0;
	counter1007: LREAL :=  0;
	counter1008: LREAL :=  0;
	counter1009: LREAL :=  0;
	counter1010: LREAL :=  0;
	counter1011: LREAL :=  0;
	counter1012: LREAL :=  0;
	counter1013: LREAL :=  0;
	counter1014: LREAL :=  0;
	counter1015: LREAL :=  0;
	counter1016: LREAL :=  0;
	counter1017: LREAL :=  0;
	counter1018: LREAL :=  0;
	counter1019: LREAL :=  0;
	counter1020: LREAL :=  0;
	counter1021: LREAL :=  0;
	counter1022: LREAL :=  0;
	counter1023: LREAL :=  0;
	counter1024: LREAL :=  0;
	counter1025: LREAL :=  0;
	counter1026: LREAL :=  0;
	counter1027: LREAL :=  0;
	counter1028: LREAL :=  0;
	counter1029: LREAL :=  0;
	counter1030: LREAL :=  0;
	counter1031: LREAL :=  0;
	counter1032: LREAL :=  0;
	counter1033: LREAL :=  0;
	counter1034: LREAL :=  0;
	counter1035: LREAL :=  0;
	counter1036: LREAL :=  0;
	counter1037: LREAL :=  0;
	counter1038: LREAL :=  0;
	counter1039: LREAL :=  0;
	counter1040: LREAL :=  0;
	counter1041: LREAL :=  0;
	counter1042: LREAL :=  0;
	counter1043: LREAL :=  0;
	counter1044: LREAL :=  0;
	counter1045: LREAL :=  0;
	counter1046: LREAL :=  0;
	counter1047: LREAL :=  0;
	counter1048: LREAL :=  0;
	counter1049: LREAL :=  0;
	counter1050: LREAL :=  0;
	counter1051: LREAL :=  0;
	counter1052: LREAL :=  0;
	counter1053: LREAL :=  0;
	counter1054: LREAL :=  0;
	counter1055: LREAL :=  0;
	counter1056: LREAL :=  0;
	counter1057: LREAL :=  0;
	counter1058: LREAL :=  0;
	counter1059: LREAL :=  0;
	counter1060: LREAL :=  0;
	counter1061: LREAL :=  0;
	counter1062: LREAL :=  0;
	counter1063: LREAL :=  0;
	counter1064: LREAL :=  0;
	counter1065: LREAL :=  0;
	counter1066: LREAL :=  0;
	counter1067: LREAL :=  0;
	counter1068: LREAL :=  0;
	counter1069: LREAL :=  0;
	counter1070: LREAL :=  0;
	counter1071: LREAL :=  0;
	counter1072: LREAL :=  0;
	counter1073: LREAL :=  0;
	counter1074: LREAL :=  0;
	counter1075: LREAL :=  0;
	counter1076: LREAL :=  0;
	counter1077: LREAL :=  0;
	counter1078: LREAL :=  0;
	counter1079: LREAL :=  0;
	counter1080: LREAL :=  0;
	counter1081: LREAL :=  0;
	counter1082: LREAL :=  0;
	counter1083: LREAL :=  0;
	counter1084: LREAL :=  0;
	counter1085: LREAL :=  0;
	counter1086: LREAL :=  0;
	counter1087: LREAL :=  0;
	counter1088: LREAL :=  0;
	counter1089: LREAL :=  0;
	counter1090: LREAL :=  0;
	counter1091: LREAL :=  0;
	counter1092: LREAL :=  0;
	counter1093: LREAL :=  0;
	counter1094: LREAL :=  0;
	counter1095: LREAL :=  0;
	counter1096: LREAL :=  0;
	counter1097: LREAL :=  0;
	counter1098: LREAL :=  0;
	counter1099: LREAL :=  0;
	counter1100: LREAL :=  0;
	counter1101: LREAL :=  0;
	counter1102: LREAL :=  0;
	counter1103: LREAL :=  0;
	counter1104: LREAL :=  0;
	counter1105: LREAL :=  0;
	counter1106: LREAL :=  0;
	counter1107: LREAL :=  0;
	counter1108: LREAL :=  0;
	counter1109: LREAL :=  0;
	counter1110: LREAL :=  0;
	counter1111: LREAL :=  0;
	counter1112: LREAL :=  0;
	counter1113: LREAL :=  0;
	counter1114: LREAL :=  0;
	counter1115: LREAL :=  0;
	counter1116: LREAL :=  0;
	counter1117: LREAL :=  0;
	counter1118: LREAL :=  0;
	counter1119: LREAL :=  0;
	counter1120: LREAL :=  0;
	counter1121: LREAL :=  0;
	counter1122: LREAL :=  0;
	counter1123: LREAL :=  0;
	counter1124: LREAL :=  0;
	counter1125: LREAL :=  0;
	counter1126: LREAL :=  0;
	counter1127: LREAL :=  0;
	counter1128: LREAL :=  0;
	counter1129: LREAL :=  0;
	counter1130: LREAL :=  0;
	counter1131: LREAL :=  0;
	counter1132: LREAL :=  0;
	counter1133: LREAL :=  0;
	counter1134: LREAL :=  0;
	counter1135: LREAL :=  0;
	counter1136: LREAL :=  0;
	counter1137: LREAL :=  0;
	counter1138: LREAL :=  0;
	counter1139: LREAL :=  0;
	counter1140: LREAL :=  0;
	counter1141: LREAL :=  0;
	counter1142: LREAL :=  0;
	counter1143: LREAL :=  0;
	counter1144: LREAL :=  0;
	counter1145: LREAL :=  0;
	counter1146: LREAL :=  0;
	counter1147: LREAL :=  0;
	counter1148: LREAL :=  0;
	counter1149: LREAL :=  0;
	counter1150: LREAL :=  0;
	counter1151: LREAL :=  0;
	counter1152: LREAL :=  0;
	counter1153: LREAL :=  0;
	counter1154: LREAL :=  0;
	counter1155: LREAL :=  0;
	counter1156: LREAL :=  0;
	counter1157: LREAL :=  0;
	counter1158: LREAL :=  0;
	counter1159: LREAL :=  0;
	counter1160: LREAL :=  0;
	counter1161: LREAL :=  0;
	counter1162: LREAL :=  0;
	counter1163: LREAL :=  0;
	counter1164: LREAL :=  0;
	counter1165: LREAL :=  0;
	counter1166: LREAL :=  0;
	counter1167: LREAL :=  0;
	counter1168: LREAL :=  0;
	counter1169: LREAL :=  0;
	counter1170: LREAL :=  0;
	counter1171: LREAL :=  0;
	counter1172: LREAL :=  0;
	counter1173: LREAL :=  0;
	counter1174: LREAL :=  0;
	counter1175: LREAL :=  0;
	counter1176: LREAL :=  0;
	counter1177: LREAL :=  0;
	counter1178: LREAL :=  0;
	counter1179: LREAL :=  0;
	counter1180: LREAL :=  0;
	counter1181: LREAL :=  0;
	counter1182: LREAL :=  0;
	counter1183: LREAL :=  0;
	counter1184: LREAL :=  0;
	counter1185: LREAL :=  0;
	counter1186: LREAL :=  0;
	counter1187: LREAL :=  0;
	counter1188: LREAL :=  0;
	counter1189: LREAL :=  0;
	counter1190: LREAL :=  0;
	counter1191: LREAL :=  0;
	counter1192: LREAL :=  0;
	counter1193: LREAL :=  0;
	counter1194: LREAL :=  0;
	counter1195: LREAL :=  0;
	counter1196: LREAL :=  0;
	counter1197: LREAL :=  0;
	counter1198: LREAL :=  0;
	counter1199: LREAL :=  0;
	counter1200: LREAL :=  0;
	counter1201: LREAL :=  0;
	counter1202: LREAL :=  0;
	counter1203: LREAL :=  0;
	counter1204: LREAL :=  0;
	counter1205: LREAL :=  0;
	counter1206: LREAL :=  0;
	counter1207: LREAL :=  0;
	counter1208: LREAL :=  0;
	counter1209: LREAL :=  0;
	counter1210: LREAL :=  0;
	counter1211: LREAL :=  0;
	counter1212: LREAL :=  0;
	counter1213: LREAL :=  0;
	counter1214: LREAL :=  0;
	counter1215: LREAL :=  0;
	counter1216: LREAL :=  0;
	counter1217: LREAL :=  0;
	counter1218: LREAL :=  0;
	counter1219: LREAL :=  0;
	counter1220: LREAL :=  0;
	counter1221: LREAL :=  0;
	counter1222: LREAL :=  0;
	counter1223: LREAL :=  0;
	counter1224: LREAL :=  0;
	counter1225: LREAL :=  0;
	counter1226: LREAL :=  0;
	counter1227: LREAL :=  0;
	counter1228: LREAL :=  0;
	counter1229: LREAL :=  0;
	counter1230: LREAL :=  0;
	counter1231: LREAL :=  0;
	counter1232: LREAL :=  0;
	counter1233: LREAL :=  0;
	counter1234: LREAL :=  0;
	counter1235: LREAL :=  0;
	counter1236: LREAL :=  0;
	counter1237: LREAL :=  0;
	counter1238: LREAL :=  0;
	counter1239: LREAL :=  0;
	counter1240: LREAL :=  0;
	counter1241: LREAL :=  0;
	counter1242: LREAL :=  0;
	counter1243: LREAL :=  0;
	counter1244: LREAL :=  0;
	counter1245: LREAL :=  0;
	counter1246: LREAL :=  0;
	counter1247: LREAL :=  0;
	counter1248: LREAL :=  0;
	counter1249: LREAL :=  0;
	counter1250: LREAL :=  0;
	counter1251: LREAL :=  0;
	counter1252: LREAL :=  0;
	counter1253: LREAL :=  0;
	counter1254: LREAL :=  0;
	counter1255: LREAL :=  0;
	counter1256: LREAL :=  0;
	counter1257: LREAL :=  0;
	counter1258: LREAL :=  0;
	counter1259: LREAL :=  0;
	counter1260: LREAL :=  0;
	counter1261: LREAL :=  0;
	counter1262: LREAL :=  0;
	counter1263: LREAL :=  0;
	counter1264: LREAL :=  0;
	counter1265: LREAL :=  0;
	counter1266: LREAL :=  0;
	counter1267: LREAL :=  0;
	counter1268: LREAL :=  0;
	counter1269: LREAL :=  0;
	counter1270: LREAL :=  0;
	counter1271: LREAL :=  0;
	counter1272: LREAL :=  0;
	counter1273: LREAL :=  0;
	counter1274: LREAL :=  0;
	counter1275: LREAL :=  0;
	counter1276: LREAL :=  0;
	counter1277: LREAL :=  0;
	counter1278: LREAL :=  0;
	counter1279: LREAL :=  0;
	counter1280: LREAL :=  0;
	counter1281: LREAL :=  0;
	counter1282: LREAL :=  0;
	counter1283: LREAL :=  0;
	counter1284: LREAL :=  0;
	counter1285: LREAL :=  0;
	counter1286: LREAL :=  0;
	counter1287: LREAL :=  0;
	counter1288: LREAL :=  0;
	counter1289: LREAL :=  0;
	counter1290: LREAL :=  0;
	counter1291: LREAL :=  0;
	counter1292: LREAL :=  0;
	counter1293: LREAL :=  0;
	counter1294: LREAL :=  0;
	counter1295: LREAL :=  0;
	counter1296: LREAL :=  0;
	counter1297: LREAL :=  0;
	counter1298: LREAL :=  0;
	counter1299: LREAL :=  0;
	counter1300: LREAL :=  0;
	counter1301: LREAL :=  0;
	counter1302: LREAL :=  0;
	counter1303: LREAL :=  0;
	counter1304: LREAL :=  0;
	counter1305: LREAL :=  0;
	counter1306: LREAL :=  0;
	counter1307: LREAL :=  0;
	counter1308: LREAL :=  0;
	counter1309: LREAL :=  0;
	counter1310: LREAL :=  0;
	counter1311: LREAL :=  0;
	counter1312: LREAL :=  0;
	counter1313: LREAL :=  0;
	counter1314: LREAL :=  0;
	counter1315: LREAL :=  0;
	counter1316: LREAL :=  0;
	counter1317: LREAL :=  0;
	counter1318: LREAL :=  0;
	counter1319: LREAL :=  0;
	counter1320: LREAL :=  0;
	counter1321: LREAL :=  0;
	counter1322: LREAL :=  0;
	counter1323: LREAL :=  0;
	counter1324: LREAL :=  0;
	counter1325: LREAL :=  0;
	counter1326: LREAL :=  0;
	counter1327: LREAL :=  0;
	counter1328: LREAL :=  0;
	counter1329: LREAL :=  0;
	counter1330: LREAL :=  0;
	counter1331: LREAL :=  0;
	counter1332: LREAL :=  0;
	counter1333: LREAL :=  0;
	counter1334: LREAL :=  0;
	counter1335: LREAL :=  0;
	counter1336: LREAL :=  0;
	counter1337: LREAL :=  0;
	counter1338: LREAL :=  0;
	counter1339: LREAL :=  0;
	counter1340: LREAL :=  0;
	counter1341: LREAL :=  0;
	counter1342: LREAL :=  0;
	counter1343: LREAL :=  0;
	counter1344: LREAL :=  0;
	counter1345: LREAL :=  0;
	counter1346: LREAL :=  0;
	counter1347: LREAL :=  0;
	counter1348: LREAL :=  0;
	counter1349: LREAL :=  0;
	counter1350: LREAL :=  0;
	counter1351: LREAL :=  0;
	counter1352: LREAL :=  0;
	counter1353: LREAL :=  0;
	counter1354: LREAL :=  0;
	counter1355: LREAL :=  0;
	counter1356: LREAL :=  0;
	counter1357: LREAL :=  0;
	counter1358: LREAL :=  0;
	counter1359: LREAL :=  0;
	counter1360: LREAL :=  0;
	counter1361: LREAL :=  0;
	counter1362: LREAL :=  0;
	counter1363: LREAL :=  0;
	counter1364: LREAL :=  0;
	counter1365: LREAL :=  0;
	counter1366: LREAL :=  0;
	counter1367: LREAL :=  0;
	counter1368: LREAL :=  0;
	counter1369: LREAL :=  0;
	counter1370: LREAL :=  0;
	counter1371: LREAL :=  0;
	counter1372: LREAL :=  0;
	counter1373: LREAL :=  0;
	counter1374: LREAL :=  0;
	counter1375: LREAL :=  0;
	counter1376: LREAL :=  0;
	counter1377: LREAL :=  0;
	counter1378: LREAL :=  0;
	counter1379: LREAL :=  0;
	counter1380: LREAL :=  0;
	counter1381: LREAL :=  0;
	counter1382: LREAL :=  0;
	counter1383: LREAL :=  0;
	counter1384: LREAL :=  0;
	counter1385: LREAL :=  0;
	counter1386: LREAL :=  0;
	counter1387: LREAL :=  0;
	counter1388: LREAL :=  0;
	counter1389: LREAL :=  0;
	counter1390: LREAL :=  0;
	counter1391: LREAL :=  0;
	counter1392: LREAL :=  0;
	counter1393: LREAL :=  0;
	counter1394: LREAL :=  0;
	counter1395: LREAL :=  0;
	counter1396: LREAL :=  0;
	counter1397: LREAL :=  0;
	counter1398: LREAL :=  0;
	counter1399: LREAL :=  0;
	counter1400: LREAL :=  0;
	counter1401: LREAL :=  0;
	counter1402: LREAL :=  0;
	counter1403: LREAL :=  0;
	counter1404: LREAL :=  0;
	counter1405: LREAL :=  0;
	counter1406: LREAL :=  0;
	counter1407: LREAL :=  0;
	counter1408: LREAL :=  0;
	counter1409: LREAL :=  0;
	counter1410: LREAL :=  0;
	counter1411: LREAL :=  0;
	counter1412: LREAL :=  0;
	counter1413: LREAL :=  0;
	counter1414: LREAL :=  0;
	counter1415: LREAL :=  0;
	counter1416: LREAL :=  0;
	counter1417: LREAL :=  0;
	counter1418: LREAL :=  0;
	counter1419: LREAL :=  0;
	counter1420: LREAL :=  0;
	counter1421: LREAL :=  0;
	counter1422: LREAL :=  0;
	counter1423: LREAL :=  0;
	counter1424: LREAL :=  0;
	counter1425: LREAL :=  0;
	counter1426: LREAL :=  0;
	counter1427: LREAL :=  0;
	counter1428: LREAL :=  0;
	counter1429: LREAL :=  0;
	counter1430: LREAL :=  0;
	counter1431: LREAL :=  0;
	counter1432: LREAL :=  0;
	counter1433: LREAL :=  0;
	counter1434: LREAL :=  0;
	counter1435: LREAL :=  0;
	counter1436: LREAL :=  0;
	counter1437: LREAL :=  0;
	counter1438: LREAL :=  0;
	counter1439: LREAL :=  0;
	counter1440: LREAL :=  0;
	counter1441: LREAL :=  0;
	counter1442: LREAL :=  0;
	counter1443: LREAL :=  0;
	counter1444: LREAL :=  0;
	counter1445: LREAL :=  0;
	counter1446: LREAL :=  0;
	counter1447: LREAL :=  0;
	counter1448: LREAL :=  0;
	counter1449: LREAL :=  0;
	counter1450: LREAL :=  0;
	counter1451: LREAL :=  0;
	counter1452: LREAL :=  0;
	counter1453: LREAL :=  0;
	counter1454: LREAL :=  0;
	counter1455: LREAL :=  0;
	counter1456: LREAL :=  0;
	counter1457: LREAL :=  0;
	counter1458: LREAL :=  0;
	counter1459: LREAL :=  0;
	counter1460: LREAL :=  0;
	counter1461: LREAL :=  0;
	counter1462: LREAL :=  0;
	counter1463: LREAL :=  0;
	counter1464: LREAL :=  0;
	counter1465: LREAL :=  0;
	counter1466: LREAL :=  0;
	counter1467: LREAL :=  0;
	counter1468: LREAL :=  0;
	counter1469: LREAL :=  0;
	counter1470: LREAL :=  0;
	counter1471: LREAL :=  0;
	counter1472: LREAL :=  0;
	counter1473: LREAL :=  0;
	counter1474: LREAL :=  0;
	counter1475: LREAL :=  0;
	counter1476: LREAL :=  0;
	counter1477: LREAL :=  0;
	counter1478: LREAL :=  0;
	counter1479: LREAL :=  0;
	counter1480: LREAL :=  0;
	counter1481: LREAL :=  0;
	counter1482: LREAL :=  0;
	counter1483: LREAL :=  0;
	counter1484: LREAL :=  0;
	counter1485: LREAL :=  0;
	counter1486: LREAL :=  0;
	counter1487: LREAL :=  0;
	counter1488: LREAL :=  0;
	counter1489: LREAL :=  0;
	counter1490: LREAL :=  0;
	counter1491: LREAL :=  0;
	counter1492: LREAL :=  0;
	counter1493: LREAL :=  0;
	counter1494: LREAL :=  0;
	counter1495: LREAL :=  0;
	counter1496: LREAL :=  0;
	counter1497: LREAL :=  0;
	counter1498: LREAL :=  0;
	counter1499: LREAL :=  0;
	counter1500: LREAL :=  0;
	counter1501: LREAL :=  0;
	counter1502: LREAL :=  0;
	counter1503: LREAL :=  0;
	counter1504: LREAL :=  0;
	counter1505: LREAL :=  0;
	counter1506: LREAL :=  0;
	counter1507: LREAL :=  0;
	counter1508: LREAL :=  0;
	counter1509: LREAL :=  0;
	counter1510: LREAL :=  0;
	counter1511: LREAL :=  0;
	counter1512: LREAL :=  0;
	counter1513: LREAL :=  0;
	counter1514: LREAL :=  0;
	counter1515: LREAL :=  0;
	counter1516: LREAL :=  0;
	counter1517: LREAL :=  0;
	counter1518: LREAL :=  0;
	counter1519: LREAL :=  0;
	counter1520: LREAL :=  0;
	counter1521: LREAL :=  0;
	counter1522: LREAL :=  0;
	counter1523: LREAL :=  0;
	counter1524: LREAL :=  0;
	counter1525: LREAL :=  0;
	counter1526: LREAL :=  0;
	counter1527: LREAL :=  0;
	counter1528: LREAL :=  0;
	counter1529: LREAL :=  0;
	counter1530: LREAL :=  0;
	counter1531: LREAL :=  0;
	counter1532: LREAL :=  0;
	counter1533: LREAL :=  0;
	counter1534: LREAL :=  0;
	counter1535: LREAL :=  0;
	counter1536: LREAL :=  0;
	counter1537: LREAL :=  0;
	counter1538: LREAL :=  0;
	counter1539: LREAL :=  0;
	counter1540: LREAL :=  0;
	counter1541: LREAL :=  0;
	counter1542: LREAL :=  0;
	counter1543: LREAL :=  0;
	counter1544: LREAL :=  0;
	counter1545: LREAL :=  0;
	counter1546: LREAL :=  0;
	counter1547: LREAL :=  0;
	counter1548: LREAL :=  0;
	counter1549: LREAL :=  0;
	counter1550: LREAL :=  0;
	counter1551: LREAL :=  0;
	counter1552: LREAL :=  0;
	counter1553: LREAL :=  0;
	counter1554: LREAL :=  0;
	counter1555: LREAL :=  0;
	counter1556: LREAL :=  0;
	counter1557: LREAL :=  0;
	counter1558: LREAL :=  0;
	counter1559: LREAL :=  0;
	counter1560: LREAL :=  0;
	counter1561: LREAL :=  0;
	counter1562: LREAL :=  0;
	counter1563: LREAL :=  0;
	counter1564: LREAL :=  0;
	counter1565: LREAL :=  0;
	counter1566: LREAL :=  0;
	counter1567: LREAL :=  0;
	counter1568: LREAL :=  0;
	counter1569: LREAL :=  0;
	counter1570: LREAL :=  0;
	counter1571: LREAL :=  0;
	counter1572: LREAL :=  0;
	counter1573: LREAL :=  0;
	counter1574: LREAL :=  0;
	counter1575: LREAL :=  0;
	counter1576: LREAL :=  0;
	counter1577: LREAL :=  0;
	counter1578: LREAL :=  0;
	counter1579: LREAL :=  0;
	counter1580: LREAL :=  0;
	counter1581: LREAL :=  0;
	counter1582: LREAL :=  0;
	counter1583: LREAL :=  0;
	counter1584: LREAL :=  0;
	counter1585: LREAL :=  0;
	counter1586: LREAL :=  0;
	counter1587: LREAL :=  0;
	counter1588: LREAL :=  0;
	counter1589: LREAL :=  0;
	counter1590: LREAL :=  0;
	counter1591: LREAL :=  0;
	counter1592: LREAL :=  0;
	counter1593: LREAL :=  0;
	counter1594: LREAL :=  0;
	counter1595: LREAL :=  0;
	counter1596: LREAL :=  0;
	counter1597: LREAL :=  0;
	counter1598: LREAL :=  0;
	counter1599: LREAL :=  0;
	counter1600: LREAL :=  0;
	counter1601: LREAL :=  0;
	counter1602: LREAL :=  0;
	counter1603: LREAL :=  0;
	counter1604: LREAL :=  0;
	counter1605: LREAL :=  0;
	counter1606: LREAL :=  0;
	counter1607: LREAL :=  0;
	counter1608: LREAL :=  0;
	counter1609: LREAL :=  0;
	counter1610: LREAL :=  0;
	counter1611: LREAL :=  0;
	counter1612: LREAL :=  0;
	counter1613: LREAL :=  0;
	counter1614: LREAL :=  0;
	counter1615: LREAL :=  0;
	counter1616: LREAL :=  0;
	counter1617: LREAL :=  0;
	counter1618: LREAL :=  0;
	counter1619: LREAL :=  0;
	counter1620: LREAL :=  0;
	counter1621: LREAL :=  0;
	counter1622: LREAL :=  0;
	counter1623: LREAL :=  0;
	counter1624: LREAL :=  0;
	counter1625: LREAL :=  0;
	counter1626: LREAL :=  0;
	counter1627: LREAL :=  0;
	counter1628: LREAL :=  0;
	counter1629: LREAL :=  0;
	counter1630: LREAL :=  0;
	counter1631: LREAL :=  0;
	counter1632: LREAL :=  0;
	counter1633: LREAL :=  0;
	counter1634: LREAL :=  0;
	counter1635: LREAL :=  0;
	counter1636: LREAL :=  0;
	counter1637: LREAL :=  0;
	counter1638: LREAL :=  0;
	counter1639: LREAL :=  0;
	counter1640: LREAL :=  0;
	counter1641: LREAL :=  0;
	counter1642: LREAL :=  0;
	counter1643: LREAL :=  0;
	counter1644: LREAL :=  0;
	counter1645: LREAL :=  0;
	counter1646: LREAL :=  0;
	counter1647: LREAL :=  0;
	counter1648: LREAL :=  0;
	counter1649: LREAL :=  0;
	counter1650: LREAL :=  0;
	counter1651: LREAL :=  0;
	counter1652: LREAL :=  0;
	counter1653: LREAL :=  0;
	counter1654: LREAL :=  0;
	counter1655: LREAL :=  0;
	counter1656: LREAL :=  0;
	counter1657: LREAL :=  0;
	counter1658: LREAL :=  0;
	counter1659: LREAL :=  0;
	counter1660: LREAL :=  0;
	counter1661: LREAL :=  0;
	counter1662: LREAL :=  0;
	counter1663: LREAL :=  0;
	counter1664: LREAL :=  0;
	counter1665: LREAL :=  0;
	counter1666: LREAL :=  0;
	counter1667: LREAL :=  0;
	counter1668: LREAL :=  0;
	counter1669: LREAL :=  0;
	counter1670: LREAL :=  0;
	counter1671: LREAL :=  0;
	counter1672: LREAL :=  0;
	counter1673: LREAL :=  0;
	counter1674: LREAL :=  0;
	counter1675: LREAL :=  0;
	counter1676: LREAL :=  0;
	counter1677: LREAL :=  0;
	counter1678: LREAL :=  0;
	counter1679: LREAL :=  0;
	counter1680: LREAL :=  0;
	counter1681: LREAL :=  0;
	counter1682: LREAL :=  0;
	counter1683: LREAL :=  0;
	counter1684: LREAL :=  0;
	counter1685: LREAL :=  0;
	counter1686: LREAL :=  0;
	counter1687: LREAL :=  0;
	counter1688: LREAL :=  0;
	counter1689: LREAL :=  0;
	counter1690: LREAL :=  0;
	counter1691: LREAL :=  0;
	counter1692: LREAL :=  0;
	counter1693: LREAL :=  0;
	counter1694: LREAL :=  0;
	counter1695: LREAL :=  0;
	counter1696: LREAL :=  0;
	counter1697: LREAL :=  0;
	counter1698: LREAL :=  0;
	counter1699: LREAL :=  0;
	counter1700: LREAL :=  0;
	counter1701: LREAL :=  0;
	counter1702: LREAL :=  0;
	counter1703: LREAL :=  0;
	counter1704: LREAL :=  0;
	counter1705: LREAL :=  0;
	counter1706: LREAL :=  0;
	counter1707: LREAL :=  0;
	counter1708: LREAL :=  0;
	counter1709: LREAL :=  0;
	counter1710: LREAL :=  0;
	counter1711: LREAL :=  0;
	counter1712: LREAL :=  0;
	counter1713: LREAL :=  0;
	counter1714: LREAL :=  0;
	counter1715: LREAL :=  0;
	counter1716: LREAL :=  0;
	counter1717: LREAL :=  0;
	counter1718: LREAL :=  0;
	counter1719: LREAL :=  0;
	counter1720: LREAL :=  0;
	counter1721: LREAL :=  0;
	counter1722: LREAL :=  0;
	counter1723: LREAL :=  0;
	counter1724: LREAL :=  0;
	counter1725: LREAL :=  0;
	counter1726: LREAL :=  0;
	counter1727: LREAL :=  0;
	counter1728: LREAL :=  0;
	counter1729: LREAL :=  0;
	counter1730: LREAL :=  0;
	counter1731: LREAL :=  0;
	counter1732: LREAL :=  0;
	counter1733: LREAL :=  0;
	counter1734: LREAL :=  0;
	counter1735: LREAL :=  0;
	counter1736: LREAL :=  0;
	counter1737: LREAL :=  0;
	counter1738: LREAL :=  0;
	counter1739: LREAL :=  0;
	counter1740: LREAL :=  0;
	counter1741: LREAL :=  0;
	counter1742: LREAL :=  0;
	counter1743: LREAL :=  0;
	counter1744: LREAL :=  0;
	counter1745: LREAL :=  0;
	counter1746: LREAL :=  0;
	counter1747: LREAL :=  0;
	counter1748: LREAL :=  0;
	counter1749: LREAL :=  0;
	counter1750: LREAL :=  0;
	counter1751: LREAL :=  0;
	counter1752: LREAL :=  0;
	counter1753: LREAL :=  0;
	counter1754: LREAL :=  0;
	counter1755: LREAL :=  0;
	counter1756: LREAL :=  0;
	counter1757: LREAL :=  0;
	counter1758: LREAL :=  0;
	counter1759: LREAL :=  0;
	counter1760: LREAL :=  0;
	counter1761: LREAL :=  0;
	counter1762: LREAL :=  0;
	counter1763: LREAL :=  0;
	counter1764: LREAL :=  0;
	counter1765: LREAL :=  0;
	counter1766: LREAL :=  0;
	counter1767: LREAL :=  0;
	counter1768: LREAL :=  0;
	counter1769: LREAL :=  0;
	counter1770: LREAL :=  0;
	counter1771: LREAL :=  0;
	counter1772: LREAL :=  0;
	counter1773: LREAL :=  0;
	counter1774: LREAL :=  0;
	counter1775: LREAL :=  0;
	counter1776: LREAL :=  0;
	counter1777: LREAL :=  0;
	counter1778: LREAL :=  0;
	counter1779: LREAL :=  0;
	counter1780: LREAL :=  0;
	counter1781: LREAL :=  0;
	counter1782: LREAL :=  0;
	counter1783: LREAL :=  0;
	counter1784: LREAL :=  0;
	counter1785: LREAL :=  0;
	counter1786: LREAL :=  0;
	counter1787: LREAL :=  0;
	counter1788: LREAL :=  0;
	counter1789: LREAL :=  0;
	counter1790: LREAL :=  0;
	counter1791: LREAL :=  0;
	counter1792: LREAL :=  0;
	counter1793: LREAL :=  0;
	counter1794: LREAL :=  0;
	counter1795: LREAL :=  0;
	counter1796: LREAL :=  0;
	counter1797: LREAL :=  0;
	counter1798: LREAL :=  0;
	counter1799: LREAL :=  0;
	counter1800: LREAL :=  0;
	counter1801: LREAL :=  0;
	counter1802: LREAL :=  0;
	counter1803: LREAL :=  0;
	counter1804: LREAL :=  0;
	counter1805: LREAL :=  0;
	counter1806: LREAL :=  0;
	counter1807: LREAL :=  0;
	counter1808: LREAL :=  0;
	counter1809: LREAL :=  0;
	counter1810: LREAL :=  0;
	counter1811: LREAL :=  0;
	counter1812: LREAL :=  0;
	counter1813: LREAL :=  0;
	counter1814: LREAL :=  0;
	counter1815: LREAL :=  0;
	counter1816: LREAL :=  0;
	counter1817: LREAL :=  0;
	counter1818: LREAL :=  0;
	counter1819: LREAL :=  0;
	counter1820: LREAL :=  0;
	counter1821: LREAL :=  0;
	counter1822: LREAL :=  0;
	counter1823: LREAL :=  0;
	counter1824: LREAL :=  0;
	counter1825: LREAL :=  0;
	counter1826: LREAL :=  0;
	counter1827: LREAL :=  0;
	counter1828: LREAL :=  0;
	counter1829: LREAL :=  0;
	counter1830: LREAL :=  0;
	counter1831: LREAL :=  0;
	counter1832: LREAL :=  0;
	counter1833: LREAL :=  0;
	counter1834: LREAL :=  0;
	counter1835: LREAL :=  0;
	counter1836: LREAL :=  0;
	counter1837: LREAL :=  0;
	counter1838: LREAL :=  0;
	counter1839: LREAL :=  0;
	counter1840: LREAL :=  0;
	counter1841: LREAL :=  0;
	counter1842: LREAL :=  0;
	counter1843: LREAL :=  0;
	counter1844: LREAL :=  0;
	counter1845: LREAL :=  0;
	counter1846: LREAL :=  0;
	counter1847: LREAL :=  0;
	counter1848: LREAL :=  0;
	counter1849: LREAL :=  0;
	counter1850: LREAL :=  0;
	counter1851: LREAL :=  0;
	counter1852: LREAL :=  0;
	counter1853: LREAL :=  0;
	counter1854: LREAL :=  0;
	counter1855: LREAL :=  0;
	counter1856: LREAL :=  0;
	counter1857: LREAL :=  0;
	counter1858: LREAL :=  0;
	counter1859: LREAL :=  0;
	counter1860: LREAL :=  0;
	counter1861: LREAL :=  0;
	counter1862: LREAL :=  0;
	counter1863: LREAL :=  0;
	counter1864: LREAL :=  0;
	counter1865: LREAL :=  0;
	counter1866: LREAL :=  0;
	counter1867: LREAL :=  0;
	counter1868: LREAL :=  0;
	counter1869: LREAL :=  0;
	counter1870: LREAL :=  0;
	counter1871: LREAL :=  0;
	counter1872: LREAL :=  0;
	counter1873: LREAL :=  0;
	counter1874: LREAL :=  0;
	counter1875: LREAL :=  0;
	counter1876: LREAL :=  0;
	counter1877: LREAL :=  0;
	counter1878: LREAL :=  0;
	counter1879: LREAL :=  0;
	counter1880: LREAL :=  0;
	counter1881: LREAL :=  0;
	counter1882: LREAL :=  0;
	counter1883: LREAL :=  0;
	counter1884: LREAL :=  0;
	counter1885: LREAL :=  0;
	counter1886: LREAL :=  0;
	counter1887: LREAL :=  0;
	counter1888: LREAL :=  0;
	counter1889: LREAL :=  0;
	counter1890: LREAL :=  0;
	counter1891: LREAL :=  0;
	counter1892: LREAL :=  0;
	counter1893: LREAL :=  0;
	counter1894: LREAL :=  0;
	counter1895: LREAL :=  0;
	counter1896: LREAL :=  0;
	counter1897: LREAL :=  0;
	counter1898: LREAL :=  0;
	counter1899: LREAL :=  0;
	counter1900: LREAL :=  0;
	counter1901: LREAL :=  0;
	counter1902: LREAL :=  0;
	counter1903: LREAL :=  0;
	counter1904: LREAL :=  0;
	counter1905: LREAL :=  0;
	counter1906: LREAL :=  0;
	counter1907: LREAL :=  0;
	counter1908: LREAL :=  0;
	counter1909: LREAL :=  0;
	counter1910: LREAL :=  0;
	counter1911: LREAL :=  0;
	counter1912: LREAL :=  0;
	counter1913: LREAL :=  0;
	counter1914: LREAL :=  0;
	counter1915: LREAL :=  0;
	counter1916: LREAL :=  0;
	counter1917: LREAL :=  0;
	counter1918: LREAL :=  0;
	counter1919: LREAL :=  0;
	counter1920: LREAL :=  0;
	counter1921: LREAL :=  0;
	counter1922: LREAL :=  0;
	counter1923: LREAL :=  0;
	counter1924: LREAL :=  0;
	counter1925: LREAL :=  0;
	counter1926: LREAL :=  0;
	counter1927: LREAL :=  0;
	counter1928: LREAL :=  0;
	counter1929: LREAL :=  0;
	counter1930: LREAL :=  0;
